# B&R Automation Studio project NAEUL004C00R13L518F00 (part 36)

#### Act_InputConfig.st
```iecst
ACTION Act_InputConfig:

	pa_tyMpProdRcp ACCESS p_ProdRcpCurrList; // Accessing the Current Product Recipe List

	tylocalMpProdRcp.In.udiRstErr := g_tyRstErrOut.udiRstErr;
	tylocalMpProdRcp.In.sPVName	  := g_tyNtParamCurr.sMpProdRcpPVNm;
	tylocalMpProdRcp.In.sFileName := g_tyNtParamCurr.sMpProdRcpFileNm;
	tylocalMpProdRcp.In.sProgNm   := g_tyNtParamCurr.sProdRcpProgNm;

	IF g_tyStartUp.bRun THEN
		tylocalMpProdRcp.In.eAct := g_tyStartUp.eMpProdRcpAct;
	ELSE
		tylocalMpProdRcp.In.eAct := g_tyUIOut.eMnlAct.eMpProdRcpAct;
	END_IF

END_ACTION
```

#### Act_Main.st
```iecst
ACTION Act_Main:

	//Set p_eAct
	IF tylocalMpProdRcp.Out.eStatus = Idle THEN
		tylocalMpProdRcp.Out.eStat	:= tylocalMpProdRcp.In.eAct;
	END_IF

	//Main
	CASE tylocalMpProdRcp.Out.eStat OF

		MpProdRcpActIdle:
			IF tylocalMpProdRcp.Out.eStatus <> Idle THEN	//Reset Data
				//Private
				fbDirCreate1(bEn := FALSE);
				fbDirCreate2(bEn := FALSE);
				fbMpRecipeRegPar(Enable := FALSE);
				fbMpRecipeXml(Enable := FALSE);
				usiStep			:= 0;

				sStatTxt	:= a_sStatText[tylocalMpProdRcp.Out.eStat];

			END_IF

			tylocalMpProdRcp.Out.eStatus	:= Idle;

		MpProdRcpActCreateDir:
			IF tylocalMpProdRcp.Out.eStatus = Idle OR tylocalMpProdRcp.Out.eStatus = Busy THEN

				tylocalMpProdRcp.Out.eStatus	:= Busy;

				sStatTxt	:= a_sStatText[tylocalMpProdRcp.Out.eStat];

				CASE usiStep OF
					0:
						fbDirCreate1(bEn := TRUE);
						IF fbDirCreate1.udiStatus = 0 THEN
							usiStep	:= 1;
						ELSIF fbDirCreate1.udiStatus < 65534 THEN
							tylocalMpProdRcp.Out.eStatus		:= Error;

							IF fbDirCreate1.udiStatus = 1908 THEN
								udiStatus	:= 10000;	//Create User Directory Error
							ELSE
								udiStatus	:= fbDirCreate1.udiStatus;
							END_IF
						END_IF

					1:
						fbDirCreate2(bEn := TRUE);
						IF fbDirCreate2.udiStatus = 0 THEN
							tylocalMpProdRcp.Out.eStatus	:= Done;
						ELSIF fbDirCreate2.udiStatus < 65534 THEN
							tylocalMpProdRcp.Out.eStatus		:= Error;

							IF fbDirCreate2.udiStatus = 1908 THEN
								udiStatus	:= 10001;	//Create Product Recipe Directory Error
							ELSE
								udiStatus	:= fbDirCreate2.udiStatus;
							END_IF
						END_IF

				END_CASE

			END_IF

		MpProdRcpActLoad:
			IF tylocalMpProdRcp.Out.eStatus = Idle OR tylocalMpProdRcp.Out.eStatus = Busy THEN

				tylocalMpProdRcp.Out.eStatus	:= Busy;

				sStatTxt	:= a_sStatText[tylocalMpProdRcp.Out.eStat];

				CASE usiStep OF
					0:
						fbMpRecipeRegPar(Enable := TRUE);

						IF (fbMpRecipeRegPar.Active = TRUE) AND (fbMpRecipeRegPar.StatusID = 0) THEN
							usiStep	:= 1;
						ELSIF fbMpRecipeRegPar.StatusID <> 0 THEN
							tylocalMpProdRcp.Out.eStatus		:= Error;
							udiStatus	:= 10002;	//MpRecipeRegPar Error While Loading
						END_IF

					1:
						fbMpRecipeXml.Load	:= TRUE;
						fbMpRecipeXml.Save	:= FALSE;
						fbMpRecipeXml(Enable := TRUE);

						IF (fbMpRecipeXml.Active = TRUE) AND (fbMpRecipeXml.CommandDone = TRUE) AND (fbMpRecipeXml.StatusID = 0) THEN
							tylocalMpProdRcp.Out.eStatus	:= Done;
							pa_tyMpProdRcp	:= a_tyMpProdRcp1;
						ELSIF fbMpRecipeXml.StatusID <> 0 THEN
							tylocalMpProdRcp.Out.eStatus		:= Error;
							udiStatus	:= 10003;	//MpRecipeXml Error While Loading
						END_IF

				END_CASE

			END_IF

		MpProdRcpActSave:
			IF tylocalMpProdRcp.Out.eStatus = Idle OR tylocalMpProdRcp.Out.eStatus = Busy THEN

				tylocalMpProdRcp.Out.eStatus	:= Busy;

				sStatTxt	:= a_sStatText[tylocalMpProdRcp.Out.eStat];

				CASE usiStep OF
					0:
						a_tyMpProdRcp1	:= pa_tyMpProdRcp;
						fbMpRecipeRegPar(Enable := TRUE);

						IF (fbMpRecipeRegPar.Active = TRUE) AND (fbMpRecipeRegPar.StatusID = 0) THEN
							usiStep	:= 1;
						ELSIF fbMpRecipeRegPar.StatusID <> 0 THEN
							tylocalMpProdRcp.Out.eStatus		:= Error;
							udiStatus	:= 10004;	//MpRecipeRegPar Error While Saving
						END_IF

					1:
						fbMpRecipeXml.Load	:= FALSE;
						fbMpRecipeXml.Save	:= TRUE;
						fbMpRecipeXml(Enable := TRUE);

						IF (fbMpRecipeXml.Active = TRUE) AND (fbMpRecipeXml.CommandDone = TRUE) AND (fbMpRecipeXml.StatusID = 0) THEN
							tylocalMpProdRcp.Out.eStatus	:= Done;
						ELSIF fbMpRecipeXml.StatusID <> 0 THEN
							tylocalMpProdRcp.Out.eStatus		:= Error;
							udiStatus	:= 10005;	//MpRecipeXml Error While Saving
						END_IF

				END_CASE

			END_IF

	END_CASE

END_ACTION
```

#### Act_OutputConfig.st
```iecst
ACTION Act_OutputConfig:

	g_tyMpProdRcp	:= tylocalMpProdRcp.Out;

END_ACTION
```

#### Cyclic.st
```iecst
PROGRAM _CYCLIC

	IF bInitialDone = FALSE THEN
		IF g_tyStartUp.bNtSettingsLoadDone = TRUE THEN
			bInitialDone	:= TRUE;
			Act_Initial;
		END_IF

	ELSE

		Act_InputConfig;
		Act_Main;
		Act_OutputConfig;
		Act_Alarm;

	END_IF

END_PROGRAM
```

### Package Logical/MagRcp - pending

### MagRcp.typ - Change By Project
```iecst
(*2020-07-24*)
(**)
(*Action*)

TYPE
	eMagRcpAction :
		(
		MagRcpActIdle,
		MagRcpActCreateDir,
		MagRcpActAddEdit,
		MagRcpActDel,
		MagRcpActGetInfo,
		MagRcpActGetList,
		MagRcpActFilter,
		MagRcpActReadCurrRcp,
		MagRcpActLoadRcp,
		MagRcpActWriteCurrRcpParam,
		MagRcpActSaveList,
		MagRcpActSort
		);
END_TYPE

(**)
(*Data*)

TYPE
	tyMagRcpParam : 	STRUCT
		sRcpNm : STRING[30];
		diTtlSlt : DINT;
		diSltToSltInUM : DINT;
		diMag1Slt1PosInUM : DINT;
		diMag2Slt1PosInUM : DINT;
		diMag3Slt1PosInUM : DINT;
		diMag1TravPosInUM : DINT;
		diMag2TravPosInUM : DINT;
		diMag3TravPosInUM : DINT;
		usiMagModel : USINT;
		sDisplayInfo : STRING[30];
		diMagMaxBrdWidth : DINT;
		dtLastModified : DATE_AND_TIME;
		bSafetyBarDisabled : BOOL;
		bMagHeightChkEn : BOOL;
	END_STRUCT;
END_TYPE
```

### MagRcp.var - Change By Project
```iecst
(*2020-07-24*)
(**)
(*Constant*)
VAR CONSTANT
	c_udiMagRcpMax : UDINT := 10;
END_VAR
(**)
(*Action & State & Status*)
VAR
	p_MagRcpStat : UDINT;
	p_MagRcpStatus : UDINT;
	p_MagRcpStatTxt : UDINT;
END_VAR
(**)
(*Alarm*)
VAR
	p_MagRcpAlmData : UDINT;
END_VAR
(**)
(*Output*)
VAR
	p_MagRcpNmExist : UDINT;
	p_MagRcpNmNotExist : UDINT;
	p_MagRcpNmEmpty : UDINT;
	p_MagRcpListFull : UDINT;
	p_MagRcpCurrList : UDINT;
	p_MagRcpFilterList : UDINT;
	p_MagRcpSortedList : UDINT;
	p_MagRcpInfoOut : UDINT;
	p_MagRcpFileNotFound : UDINT;
	p_MagRcpCurrRcp : UDINT;
	p_MagRcpCurrRcpNm : UDINT;
	p_MagRcpCurrRcpTtlSlt : UDINT;
	p_MagRcpCurrRcpSltToSlt : UDINT;
	p_MagRcpCurrRcpMag1Slt1Pos : UDINT;
	p_MagRcpCurrRcpMag2Slt1Pos : UDINT;
	p_MagRcpCurrRcpMag3Slt1Pos : UDINT;
	p_MagRcpCurrRcpMag1TravPos : UDINT;
	p_MagRcpCurrRcpMag2TravPos : UDINT;
	p_MagRcpCurrRcpMag3TravPos : UDINT;
	p_MagRcpCurrRcpDisplayInfo : UDINT;
	p_MagRcpCurrRcpMagMaxBrdWidth : UDINT;
	p_MagRcpCurrRcpLastModified : UDINT;
	p_MagRcpCurrRcpMagModel : UDINT;
	p_MagRcpCurrRcpSBarDisabled : UDINT;
	p_MagRcpCurrRcpMagHeightChkEn : UDINT;
END_VAR
(**)
```

### Program Logical/MagRcp/MagRcp (IEC) - 1.00.0 - NtRecipe v5.00.0 , NtFileIO v5.00.0

#### InputRef.var
```iecst
(*2019-05-07*)
(**)
(*General*)
VAR
	p_eAct : REFERENCE TO eMagRcpAction;
	p_udiMax : REFERENCE TO UDINT;
	p_udiRstErr : REFERENCE TO UDINT;
	p_bPrep : REFERENCE TO BOOL;
	p_bDis : REFERENCE TO BOOL;
END_VAR
(**)
(*Configuration*)
VAR
	p_dtCurrDT : REFERENCE TO DATE_AND_TIME;
	p_sSearch : REFERENCE TO STRING[30];
	p_tyInfoIn : REFERENCE TO tyMagRcpParam;
	p_tyCurrRcpWr : REFERENCE TO tyMagRcpParam;
	p_sListFileName : REFERENCE TO STRING[80];
	p_sSingleFileName : REFERENCE TO STRING[80];
	p_sProgNm : REFERENCE TO STRING[15];
	p_bNtSettingsLoadDone : REFERENCE TO BOOL;
	p_eLinkLCSMngRcpMagRcpAct : REFERENCE TO eMagRcpAction;
	p_bLinkNtParamLCSManageRcpPrep : REFERENCE TO BOOL;
	p_bLinkMcParamLCSManageRcpEn : REFERENCE TO BOOL;
	p_eLinkUIMagRcpAct : REFERENCE TO eMagRcpAction;
END_VAR
```

#### InputRef_Link.var
```iecst
(*2019-03-25*)
(**)
VAR
	rSltToSlt : REAL;
	sSltToSlt : STRING[30];
	sTtlSlt : STRING[30];
	p_bLinkStartupRun : REFERENCE TO BOOL;
END_VAR
```

#### Local.var
```iecst
(*2019-05-09*)
(**)
(*Local Action, State & Status*)
VAR
	eAct : eMagRcpAction := MagRcpActIdle;
	eStat : eMagRcpAction := MagRcpActIdle;
	eStatus : eFBStatus := Idle;
	udiStatus : UDINT := 0;
	sStatTxt : STRING[200] := '';
	a_sStatText : ARRAY[0..50] OF STRING[200] := ['Idling','Creating Directory','Adding and Editing Files','Deleting Files','Get Info','Get List','Filtering Files','Reading Current Recipe','Loading Current Recipe','Writing Current Recipe Parameter','Saving List',40('')];
END_VAR
(**)
(*Local Alarm*)
VAR
	tyAlmData : tyAlmDat;
	a_tyAlmText : ARRAY[10000..10099] OF tyAlmTxt := [(sAlmText:='Create User Directory Error',sRcyText:='Unable To Create User Directory. Please Contact Nutek For A Possible Solution'),(sAlmText:='Create Magazine Recipe Directory Error',sRcyText:='Unable To Create Magazine Recipe Directory. Please Contact Nutek For A Possible Solution'),(sAlmText:='File Open Error While Adding & Editing',sRcyText:='An Error Was Encountered While Trying To Open File. Please Contact Nutek For A Possible Solution.'),(sAlmText:='File Create Error While Adding & Editing',sRcyText:='An Error Was Encountered While Trying To Create File. Please Contact Nutek For A Possible Solution.'),(sAlmText:='File Write Error While Adding & Editing',sRcyText:='An Error Was Encountered While Trying To Write File. Please Contact Nutek For A Possible Solution.'),(sAlmText:='File Close Error While Adding & Editing',sRcyText:='An Error Was Encountered While Trying To Close File. Please Contact Nutek For A Possible Solution.'),(sAlmText:='File Open Error While Deleting',sRcyText:='An Error Was Encountered While Trying To Open File. Please Contact Nutek For A Possible Solution.'),(sAlmText:='File Create Error While Deleting',sRcyText:='An Error Was Encountered While Trying To Create File. Please Contact Nutek For A Possible Solution.'),(sAlmText:='File Write Error While Deleting',sRcyText:='An Error Was Encountered While Trying To Write File. Please Contact Nutek For A Possible Solution.'),(sAlmText:='File Close Error While Deleting',sRcyText:='An Error Was Encountered While Trying To Close File. Please Contact Nutek For A Possible Solution.'),(sAlmText:='File Open Error While Getting List',sRcyText:='An Error Was Encountered While Trying To Open File. Please Contact Nutek For A Possible Solution.'),(sAlmText:='File Read Error While Getting List',sRcyText:='An Error Was Encountered While Trying To Read File. Please Contact Nutek For A Possible Solution.'),(sAlmText:='File Close Error While Getting List',sRcyText:='An Error Was Encountered While Trying To Close File. Please Contact Nutek For A Possible Solution.'),(sAlmText:='Directory Does Not Exist While Adding & Editing',sRcyText:='The Directory Does Not Exist.Please Contact Nutek For A Possible Solution.'),(sAlmText:='Directory Does Not Exist While Deleting',sRcyText:='The Directory Does Not Exist.Please Contact Nutek For A Possible Solution.'),(sAlmText:='File Open Error While Loading Current Recipe',sRcyText:='An Error Was Encountered While Trying To Open File. Please Contact Nutek For A Possible Solution.'),(sAlmText:='File Create Error While Loading Current Recipe',sRcyText:='An Error Was Encountered While Trying To Create File. Please Contact Nutek For A Possible Solution.'),(sAlmText:='File Write Error While Loading Current Recipe',sRcyText:='An Error Was Encountered While Trying To Write File. Please Contact Nutek For A Possible Solution.'),(sAlmText:='File Close Error While Loading Current Recipe',sRcyText:='An Error Was Encountered While Trying To Close File. Please Contact Nutek For A Possible Solution.'),(sAlmText:='Directory Does Not Exist While Loading Current Recipe',sRcyText:='The Directory Does Not Exist.Please Contact Nutek For A Possible Solution.'),(sAlmText:='File Open Error While Reading Current Recipe',sRcyText:='An Error Was Encountered While Trying To Open File. Please Contact Nutek For A Possible Solution.'),(sAlmText:='File Read Error While Reading Current Recipe',sRcyText:='An Error Was Encountered While Trying To Read File. Please Contact Nutek For A Possible Solution.'),(sAlmText:='File Close Error While Reading Current Recipe',sRcyText:='An Error Was Encountered While Trying To Close File. Please Contact Nutek For A Possible Solution.'),(sAlmText:='File Open Error While Writing Current Recipe Parameter',sRcyText:='An Error Was Encountered While Trying To Open File. Please Contact Nutek For A Possible Solution.'),(sAlmText:='File Create Error While Writing Current Recipe Parameter',sRcyText:='An Error Was Encountered While Trying To Create File. Please Contact Nutek For A Possible Solution.'),(sAlmText:='File Write Error While Writing Current Recipe Parameter',sRcyText:='An Error Was Encountered While Trying To Write File. Please Contact Nutek For A Possible Solution.'),(sAlmText:='File Close Error While Writing Current Recipe Parameter',sRcyText:='An Error Was Encountered While Trying To Close File. Please Contact Nutek For A Possible Solution.'),(sAlmText:='Directory Does Not Exist While Writing Current Recipe Parameter',sRcyText:='The Directory Does Not Exist.Please Contact Nutek For A Possible Solution.'),(sAlmText:='File Open Error While Saving List',sRcyText:='An Error Was Encountered While Trying To Open File. Please Contact Nutek For A Possible Solution.'),(sAlmText:='File Create Error While Saving List',sRcyText:='An Error Was Encountered While Trying To Create File. Please Contact Nutek For A Possible Solution.'),(sAlmText:='File Write Error While Saving List',sRcyText:='An Error Was Encountered While Trying To Write File. Please Contact Nutek For A Possible Solution.'),(sAlmText:='File Close Error While Saving List',sRcyText:='An Error Was Encountered While Trying To Close File. Please Contact Nutek For A Possible Solution.'),(sAlmText:='Directory Does Not Exist While Saving List',sRcyText:='The Directory Does Not Exist.Please Contact Nutek For A Possible Solution.'),67(0)];
END_VAR
(**)
(*Local Output*)
VAR
	bNmExist : BOOL;
	bNmNotExist : BOOL;
	bNmEmpty : BOOL;
	bListFull : BOOL;
	a_tyCurrList : ARRAY[1..c_udiMagRcpMax] OF tyMagRcpParam;
	a_tyFilterList : ARRAY[1..c_udiMagRcpMax] OF tyMagRcpParam;
	a_tySortList : ARRAY[1..c_udiMagRcpMax] OF tyMagRcpParam;
	tyTempList : tyMagRcpParam;
	tyInfoOut : tyMagRcpParam;
	bFileNotFound : BOOL;
	tyCurrRcp : tyMagRcpParam;
END_VAR
(**)
(*Local Input*)
VAR
	udiRstErr : UDINT := 0;
	bPrep : BOOL := TRUE;
	bDis : BOOL := FALSE;
	dtCurrDT : DATE_AND_TIME;
	sSearch : STRING[30] := '';
	tyInfoIn : tyMagRcpParam;
	tyCurrRcpWr : tyMagRcpParam;
	sListFileName : STRING[80] := 'MagazineRecipeList.dat';
	sSingleFileName : STRING[80] := 'MagazineRecipe.dat';
	sProgNm : STRING[15] := 'MagRcp';
	bNtSettingsLoadDone : BOOL := TRUE;
	udiSortCurrenTotalCntr : UDINT;
	iSortCurrentInnerCntr : INT;
	iSortCurrentOuterCntr : INT;
	iTotalRcp : INT;
	i : {REDUND_UNREPLICABLE} INT;
	udi : UDINT;
	sDebug : STRING[300];
	tyTempRecipe : tyMagRcpParam;
END_VAR
(**)
(*Local*)
VAR
	bRstErr : BOOL;
	udiRstErrOld : UDINT;
	bInitDone : BOOL;
	bInitialDone : BOOL;
	usiStep : USINT;
	udiAddStatus : UDINT;
	a_tyListTemp : ARRAY[1..c_udiMagRcpMax] OF tyMagRcpParam;
	fbDirCreate1 : fbDirCreate;
	fbDirCreate2 : fbDirCreate;
	fbFileReadList : fbFileFullRead;
	fbFileWriteList : fbFileFullWrite;
	fbFileReadSingle : fbFileFullRead;
	fbFileWriteSingle : fbFileFullWrite;
	fbFileLoadSingle : fbFileFullWrite;
	iFilterCtr : INT;
	udiModuleNum : UDINT := 4901;
END_VAR
```

#### Act_Action.st
```iecst
(** 2019-03-25 **)
ACTION Act_Action:

	//Reset Error
	IF (eStatus = Error) AND bRstErr THEN
		p_eAct	:= MagRcpActIdle;
		eStat	:= MagRcpActIdle;
	END_IF

	//Reset Done
	IF eStatus = Done AND p_eAct = MagRcpActIdle THEN
		eStat	:= MagRcpActIdle;
	END_IF

	//Set p_eAct
	IF eStatus = Idle THEN
		eStat	:= p_eAct;
	END_IF

END_ACTION
```

#### Act_Alarm.st
```iecst
(** 2019-03-25 **)
ACTION Act_Alarm:

	//Error
	IF EDGEPOS(eStatus = Error) THEN

		tyAlmData.sProgNm		:= p_sProgNm;
		tyAlmData.udiCode		:= udiStatus;
		tyAlmData.eSeverity		:= AlmSeverityError;
		tyAlmData.udiRunTime	:= tyAlmData.udiRunTime + 1;
		tyAlmData.bAlm			:= TRUE;
		tyAlmData.udiModuleNum  := udiModuleNum;
		g_sMagRcpProgNm			:= p_sProgNm;

		//Get Error Message
		IF tyAlmData.udiCode < 10000 OR tyAlmData.udiCode > 10099 THEN
			tyAlmData.sAlmMsg	:= 'Unknown';
			tyAlmData.sRcyMsg	:= 'Unknown';
		ELSE
			tyAlmData.sAlmMsg	:= a_tyAlmText[tyAlmData.udiCode].sAlmText;
			tyAlmData.sRcyMsg	:= a_tyAlmText[tyAlmData.udiCode].sRcyText;
		END_IF

		sStatTxt	:= tyAlmData.sAlmMsg;

	ELSIF bRstErr AND (tyAlmData.udiCode <> 0) THEN

		tyAlmData.udiCode	:= 0;
		tyAlmData.eSeverity	:= AlmSeverityNA;
		tyAlmData.sAlmMsg	:= '';
		tyAlmData.sRcyMsg	:= '';
		tyAlmData.bAlm			:= FALSE;
		sStatTxt	:= a_sStatText[eStat];

	END_IF

END_ACTION
```

#### Act_InitGlobal.st
```iecst
(** 2019-03-25 **)
ACTION Act_InitGlobal:

	(* Always Change If Project Change *)

	//Pass Data To Link
	p_bLinkStartupRun ACCESS p_StartupRun;

	//Pass Data To Internal Use
	p_udiRstErr ACCESS p_RstErrReset;
	p_dtCurrDT ACCESS p_TimeCurrDT;
	p_sSearch ACCESS p_UIMagRcpSearch;
	//p_tyInfoIn ACCESS p_UIMagRcpInfoIn;
	p_sListFileName ACCESS p_NtParamMagRcpListFileNm;
	p_sSingleFileName ACCESS p_NtParamMagRcpSingleFileNm;
	p_sProgNm ACCESS p_NtParamMagRcpProgNm;
	p_bNtSettingsLoadDone ACCESS p_StartupNtSettingsLoadDone;
	p_eLinkLCSMngRcpMagRcpAct ACCESS p_LCSMngRcpMagRcpAct;
	p_bLinkNtParamLCSManageRcpPrep ACCESS p_NtParamLCSManageRcpPrep;
	p_bLinkMcParamLCSManageRcpEn ACCESS p_McParamLCSManageRcpEn;
	p_eLinkUIMagRcpAct ACCESS p_UIMagRcpAct;
	(* Always Change If Project Change *)

END_ACTION
```

#### Act_Initial.st
```iecst
(** 2019-05-07 **)
ACTION Act_Initial:

	//Initial
	sStatTxt	:= a_sStatText[eStat];

	fbDirCreate1.sDevice	:= 'F';
	fbDirCreate1.sDirName	:= 'User';
	fbDirCreate1(bEn := FALSE);

	fbDirCreate2.sDevice	:= 'User';
	fbDirCreate2.sDirName	:= 'MagazineRecipe';
	fbDirCreate2(bEn := FALSE);

	fbFileReadList.sDevice			:= 'MagRcp';
	fbFileReadList.sFile			:= p_sListFileName;
	fbFileReadList.udiOffset		:= 0;
	fbFileReadList.p_Dest			:= ADR(a_tyCurrList);
	fbFileReadList.udiLen			:= SIZEOF(a_tyCurrList);
	fbFileReadList(bEn := FALSE);

	fbFileWriteList.sDevice			:= 'MagRcp';
	fbFileWriteList.sFile			:= p_sListFileName;
	fbFileWriteList.udiOffset		:= 0;
	fbFileWriteList.p_Src			:= ADR(a_tyListTemp);
	fbFileWriteList.udiLen			:= SIZEOF(a_tyListTemp);
	fbFileWriteList.udiOption		:= 0;
	fbFileWriteList(bEn := FALSE);

	fbFileReadSingle.sDevice		:= 'MagRcp';
	fbFileReadSingle.sFile			:= p_sSingleFileName;
	fbFileReadSingle.udiOffset		:= 0;
	fbFileReadSingle.p_Dest			:= ADR(tyCurrRcp);
	fbFileReadSingle.udiLen			:= SIZEOF(tyCurrRcp);
	fbFileReadSingle(bEn := FALSE);

	fbFileLoadSingle.sDevice		:= 'MagRcp';
	fbFileLoadSingle.sFile			:= p_sSingleFileName;
	fbFileLoadSingle.udiOffset		:= 0;
	fbFileLoadSingle.p_Src			:= ADR(tyCurrRcp);
	fbFileLoadSingle.udiLen			:= SIZEOF(tyCurrRcp);
	fbFileLoadSingle.udiOption		:= 0;
	fbFileLoadSingle(bEn := FALSE);

	fbFileWriteSingle.sDevice		:= 'MagRcp';
	fbFileWriteSingle.sFile			:= p_sSingleFileName;
	fbFileWriteSingle.udiOffset		:= 0;
	fbFileWriteSingle.p_Src			:= ADR(p_tyCurrRcpWr);
	fbFileWriteSingle.udiLen		:= SIZEOF(p_tyCurrRcpWr);
	fbFileWriteSingle.udiOption		:= 0;
	fbFileWriteSingle(bEn := FALSE);

END_ACTION
```

#### Act_InitLocal.st
```iecst
(** 2019-05-07 **)
ACTION Act_InitLocal:

	//Input Reference Link To Local Variable
	p_eAct ACCESS ADR(eAct);
	p_udiMax ACCESS ADR(c_udiMagRcpMax);
	p_udiRstErr ACCESS ADR(udiRstErr);
	p_bPrep ACCESS ADR(bPrep);
	p_bDis ACCESS ADR(bDis);
	p_dtCurrDT ACCESS ADR(dtCurrDT);
	p_sSearch ACCESS ADR(sSearch);
	p_tyInfoIn ACCESS ADR(tyInfoIn);
	p_tyCurrRcpWr ACCESS ADR(tyCurrRcpWr);
	p_sListFileName ACCESS ADR(sListFileName);
	p_sSingleFileName ACCESS ADR(sSingleFileName);
	p_sProgNm ACCESS ADR(sProgNm);
	p_bNtSettingsLoadDone ACCESS ADR(bNtSettingsLoadDone);

END_ACTION
```

#### Act_Link.st
```iecst
(** 2019-03-29 **)
ACTION Act_Link:

	IF p_eAct = MagRcpActAddEdit THEN

		rSltToSlt	:= DINT_TO_REAL(p_tyInfoIn.diSltToSltInUM);
		rSltToSlt	:= rSltToSlt / 1000;
		sSltToSlt	:= REAL_TO_STRING(rSltToSlt);
		sTtlSlt		:= DINT_TO_STRING(p_tyInfoIn.diTtlSlt);

		p_tyInfoIn.sDisplayInfo	:= sSltToSlt;
		p_tyInfoIn.sDisplayInfo	:= CONCAT(p_tyInfoIn.sDisplayInfo , ' | ');
		p_tyInfoIn.sDisplayInfo	:= CONCAT(p_tyInfoIn.sDisplayInfo , sTtlSlt);

	END_IF

END_ACTION
```

#### Act_LinkAction.st
```iecst
(** 2019-03-29 **)
ACTION Act_LinkAction:

	IF p_bLinkStartupRun = TRUE THEN
		p_eAct ACCESS p_StartupMagRcpAct;
	ELSE

		IF p_bLinkNtParamLCSManageRcpPrep AND p_bLinkMcParamLCSManageRcpEn THEN
			IF p_eLinkLCSMngRcpMagRcpAct <> MagRcpActIdle THEN
				p_eAct ACCESS p_LCSMngRcpMagRcpAct;
				p_tyInfoIn ACCESS p_LCSMngRcpMagRcpInfoIn;
			ELSIF p_eLinkUIMagRcpAct <> MagRcpActIdle THEN
				p_eAct ACCESS p_UIMagRcpAct;
				p_tyInfoIn ACCESS p_UIMagRcpInfoIn;

				p_tyInfoIn.dtLastModified	:= p_dtCurrDT;
			END_IF
		ELSE
			p_eAct ACCESS p_UIMagRcpAct;
			p_tyInfoIn ACCESS p_UIMagRcpInfoIn;

			p_tyInfoIn.dtLastModified	:= p_dtCurrDT;
		END_IF
	END_IF

END_ACTION
```

#### Act_Main.st
```iecst
(** 2019-05-09 **)
ACTION Act_Main:

	//Main
	CASE eStat OF

		MagRcpActIdle:
			IF eStatus <> Idle THEN	//Reset Data
				//Private
				fbDirCreate1(bEn := FALSE);
				fbDirCreate2(bEn := FALSE);
				fbFileReadList(bEn := FALSE);
				fbFileWriteList(bEn := FALSE);
				fbFileReadSingle(bEn := FALSE);
				fbFileWriteSingle(bEn := FALSE);
				fbFileLoadSingle(bEn := FALSE);
				usiStep			:= 0;
				udiAddStatus	:= 0;

				bNmExist		:= FALSE;
				bNmNotExist		:= FALSE;
				bNmEmpty		:= FALSE;
				bListFull		:= FALSE;
				bFileNotFound	:= FALSE;
				iTotalRcp		:= 0;

				memset(ADR(tyTempRecipe), 0 , SIZEOF(tyTempRecipe));

				sStatTxt	:= a_sStatText[eStat];

			END_IF

			eStatus	:= Idle;

		MagRcpActCreateDir:
			IF eStatus = Idle OR eStatus = Busy THEN

				eStatus	:= Busy;

				sStatTxt	:= a_sStatText[eStat];

				CASE usiStep OF
					0:
						fbDirCreate1(bEn := TRUE);
						IF fbDirCreate1.udiStatus = 0 THEN
							usiStep	:= 1;
						ELSIF fbDirCreate1.udiStatus < 65534 THEN
							eStatus		:= Error;

							IF fbDirCreate1.udiStatus = 1908 THEN
								udiStatus	:= 10000;	//Create User Directory Error
							ELSE
								udiStatus	:= fbDirCreate1.udiStatus;
							END_IF
						END_IF

					1:
						fbDirCreate2(bEn := TRUE);
						IF fbDirCreate2.udiStatus = 0 THEN
							eStatus	:= Done;
						ELSIF fbDirCreate2.udiStatus < 65534 THEN
							eStatus		:= Error;

							IF fbDirCreate2.udiStatus = 1908 THEN
								udiStatus	:= 10001;	//Create Magazine Recipe Directory Error
							ELSE
								udiStatus	:= fbDirCreate2.udiStatus;
							END_IF
						END_IF

				END_CASE

			END_IF

		MagRcpActAddEdit:
			IF eStatus = Idle OR eStatus = Busy THEN

				eStatus	:= Busy;

				sStatTxt	:= a_sStatText[eStat];

				CASE usiStep OF
					0:	//Edit Recipe
						udiAddStatus	:= fRecipeAddEdit(ADR(p_tyInfoIn) , ADR(a_tyListTemp) , SIZEOF(a_tyListTemp[1]) , ADR(a_tyListTemp[1].sRcpNm) , SIZEOF(a_tyListTemp[1].sRcpNm) , p_udiMax);

						IF udiAddStatus = 1600 THEN	//Recipe Name Empty
							bNmEmpty	:= TRUE;
							eStatus		:= Done;

						ELSIF udiAddStatus = 1601 THEN	//Recipe Full
							bListFull	:= TRUE;
							eStatus		:= Done;

						ELSIF udiAddStatus = 0 THEN	//OK
							usiStep	:= 1;

						END_IF

					1:	//Write Into File
						fbFileWriteList(bEn := TRUE);

						IF fbFileWriteList.udiStatus = 0 THEN
							a_tyCurrList	:= a_tyListTemp;
							eStatus			:= Done;

						ELSIF fbFileWriteList.udiStatus < 65534 THEN
							a_tyListTemp	:= a_tyCurrList;
							eStatus			:= Error;

							IF fbFileWriteList.udiStatus = 1900 THEN
								udiStatus	:= 10002;	//File Open Error While Adding & Editing
							ELSIF fbFileWriteList.udiStatus = 1901 THEN
								udiStatus	:= 10003;	//File Create Error While Adding & Editing
							ELSIF fbFileWriteList.udiStatus = 1903 THEN
								udiStatus	:= 10004;	//File Write Error While Adding & Editing
							ELSIF fbFileWriteList.udiStatus = 1904 THEN
								udiStatus	:= 10005;	//File Close Error While Adding & Editing
							ELSIF fbFileWriteList.udiStatus = 1914 THEN
								udiStatus	:= 10013;	//Directory Does Not Exist While Adding & Editing
							ELSE
								udiStatus	:= fbFileWriteList.udiStatus;
							END_IF
						END_IF

				END_CASE

			END_IF

		MagRcpActDel:
			IF eStatus = Idle OR eStatus = Busy THEN

				eStatus	:= Busy;

				sStatTxt	:= a_sStatText[eStat];

				CASE usiStep OF
					0:	//Delete Recipe
						udiAddStatus	:= fRecipeDelete(ADR(p_tyInfoIn) , ADR(a_tyListTemp) , SIZEOF(a_tyListTemp[1]) , ADR(a_tyListTemp[1].sRcpNm) , SIZEOF(a_tyListTemp[1].sRcpNm) , p_udiMax);

						IF udiAddStatus = 1600 THEN	//Recipe Name Empty
							bNmEmpty	:= TRUE;
							eStatus		:= Done;

						ELSIF udiAddStatus = 1603 THEN	//Recipe Not Exist
							bNmNotExist	:= TRUE;
							eStatus		:= Done;

						ELSIF udiAddStatus = 0 THEN	//OK
							usiStep	:= 1;

						END_IF

					1:	//Write Into File
						fbFileWriteList(bEn := TRUE);

						IF fbFileWriteList.udiStatus = 0 THEN
							a_tyCurrList	:= a_tyListTemp;
							eStatus			:= Done;

						ELSIF fbFileWriteList.udiStatus < 65534 THEN
							a_tyListTemp	:= a_tyCurrList;
							eStatus			:= Error;

							IF fbFileWriteList.udiStatus = 1900 THEN
								udiStatus	:= 10006;	//File Open Error While Deleting
							ELSIF fbFileWriteList.udiStatus = 1901 THEN
								udiStatus	:= 10007;	//File Create Error While Deleting
							ELSIF fbFileWriteList.udiStatus = 1903 THEN
								udiStatus	:= 10008;	//File Write Error While Deleting
							ELSIF fbFileWriteList.udiStatus = 1904 THEN
								udiStatus	:= 10009;	//File Close Error While Deleting
							ELSIF fbFileWriteList.udiStatus = 1914 THEN
								udiStatus	:= 10014;	//Directory Does Not Exist While Deleting
							ELSE
								udiStatus	:= fbFileWriteList.udiStatus;
							END_IF
						END_IF

				END_CASE

			END_IF

		MagRcpActGetInfo:
			IF eStatus = Idle OR eStatus = Busy THEN

				sStatTxt	:= a_sStatText[eStat];

				IF p_tyInfoIn.sRcpNm = '' THEN
					bNmEmpty	:= TRUE;
					bNmNotExist	:= TRUE;
				ELSE
					bNmNotExist	:= (fRecipeGetInfo(p_tyInfoIn.sRcpNm , ADR(tyInfoOut) , ADR(a_tyCurrList) , SIZEOF(a_tyCurrList[1]) , ADR(a_tyCurrList[1].sRcpNm) , SIZEOF(a_tyCurrList[1].sRcpNm) , p_udiMax)) = 0;
				END_IF

				eStatus	:= Done;

			END_IF

		MagRcpActGetList:
			IF eStatus = Idle OR eStatus = Busy THEN

				eStatus	:= Busy;

				sStatTxt	:= a_sStatText[eStat];

				fbFileReadList(bEn := TRUE);
				IF fbFileReadList.udiStatus = 0 THEN
					a_tyListTemp	:= a_tyCurrList;
					eStatus			:= Done;

				ELSIF fbFileReadList.udiStatus < 65534 THEN
					eStatus		:= Error;

					IF fbFileReadList.udiStatus = 1900 THEN
						udiStatus	:= 10010;	//File Open Error While Getting List
					ELSIF fbFileReadList.udiStatus = 1902 THEN
						udiStatus	:= 10011;	//File Read Error While Getting List
					ELSIF fbFileReadList.udiStatus = 1904 THEN
						udiStatus	:= 10012;	//File Close Error While Getting List
					ELSIF fbFileReadList.udiStatus = 1915 THEN
						bFileNotFound	:= TRUE;
						eStatus			:= Done;
					ELSE
						udiStatus	:= fbFileReadList.udiStatus;
					END_IF
				END_IF

			END_IF

		MagRcpActFilter:
			IF eStatus = Idle OR eStatus = Busy THEN

				sStatTxt	:= a_sStatText[eStat];

				CASE usiStep OF
					0:
						fRecipeFilter(p_sSearch , ADR(a_tyFilterList) , ADR(a_tyCurrList) , SIZEOF(a_tyCurrList[1]) , ADR(a_tyCurrList[1].sRcpNm) ,
						SIZEOF(a_tyCurrList[1].sRcpNm) , p_udiMax, 0, 499, iFilterCtr);
						usiStep := 1;
					1:
						fRecipeFilter(p_sSearch , ADR(a_tyFilterList) , ADR(a_tyCurrList) , SIZEOF(a_tyCurrList[1]) , ADR(a_tyCurrList[1].sRcpNm) ,
						SIZEOF(a_tyCurrList[1].sRcpNm) , p_udiMax, 500, 999, iFilterCtr);
						usiStep := 2;
					2:
						fRecipeFilter(p_sSearch , ADR(a_tyFilterList) , ADR(a_tyCurrList) , SIZEOF(a_tyCurrList[1]) , ADR(a_tyCurrList[1].sRcpNm) ,
						SIZEOF(a_tyCurrList[1].sRcpNm) , p_udiMax, 1000, 1499, iFilterCtr);
						usiStep := 3;
					3:
						fRecipeFilter(p_sSearch , ADR(a_tyFilterList) , ADR(a_tyCurrList) , SIZEOF(a_tyCurrList[1]) , ADR(a_tyCurrList[1].sRcpNm) ,
						SIZEOF(a_tyCurrList[1].sRcpNm) , p_udiMax, 1500, 1999, iFilterCtr);
						eStatus := Done;

				END_CASE

				eStatus	:= Done;

			END_IF

		MagRcpActLoadRcp:
			IF eStatus = Idle OR eStatus = Busy THEN

				sStatTxt	:= a_sStatText[eStat];

				CASE usiStep OF
					0:	//Get Recipe
						IF p_tyInfoIn.sRcpNm = '' THEN
							bNmEmpty	:= TRUE;
							bNmNotExist	:= TRUE;

							eStatus	:= Done;
						ELSE
							bNmNotExist	:= (fRecipeGetInfo(p_tyInfoIn.sRcpNm , ADR(tyCurrRcp) , ADR(a_tyCurrList) , SIZEOF(a_tyCurrList[1]) , ADR(a_tyCurrList[1].sRcpNm) , SIZEOF(a_tyCurrList[1].sRcpNm) , p_udiMax)) = 0;
							IF bNmNotExist = TRUE THEN
								eStatus	:= Done;
							ELSE
								usiStep	:= 1;
							END_IF
						END_IF

					1:	//Write Into File
						fbFileLoadSingle(bEn := TRUE);

						IF fbFileLoadSingle.udiStatus = 0 THEN
							eStatus			:= Done;
						ELSIF fbFileLoadSingle.udiStatus < 65534 THEN
							eStatus			:= Error;

							IF fbFileLoadSingle.udiStatus = 1900 THEN
								udiStatus	:= 10015;	//File Open Error While Loading Current Recipe
							ELSIF fbFileLoadSingle.udiStatus = 1901 THEN
								udiStatus	:= 10016;	//File Create Error While Loading Current Recipe
							ELSIF fbFileLoadSingle.udiStatus = 1903 THEN
								udiStatus	:= 10017;	//File Write Error While Loading Current Recipe
							ELSIF fbFileLoadSingle.udiStatus = 1904 THEN
								udiStatus	:= 10018;	//File Close Error While Loading Current Recipe
							ELSIF fbFileLoadSingle.udiStatus = 1914 THEN
								udiStatus	:= 10019;	//Directory Does Not Exist While Loading Current Recipe
							ELSE
								udiStatus	:= fbFileLoadSingle.udiStatus;
							END_IF
						END_IF

				END_CASE

			END_IF

		MagRcpActReadCurrRcp:
			IF eStatus = Idle OR eStatus = Busy THEN

				eStatus	:= Busy;

				sStatTxt	:= a_sStatText[eStat];

				fbFileReadSingle(bEn := TRUE);
				IF fbFileReadSingle.udiStatus = 0 THEN
					eStatus	:= Done;

				ELSIF fbFileReadSingle.udiStatus < 65534 THEN
					eStatus		:= Error;

					IF fbFileReadSingle.udiStatus = 1900 THEN
						udiStatus	:= 10020;	//File Open Error While Reading Current Recipe
					ELSIF fbFileReadSingle.udiStatus = 1902 THEN
						udiStatus	:= 10021;	//File Read Error While Reading Current Recipe
					ELSIF fbFileReadSingle.udiStatus = 1904 THEN
						udiStatus	:= 10022;	//File Close Error While Reading Current Recipe
					ELSIF fbFileReadSingle.udiStatus = 1915 THEN
						bFileNotFound	:= TRUE;
						eStatus			:= Done;
					ELSE
						udiStatus	:= fbFileReadSingle.udiStatus;
					END_IF
				END_IF

			END_IF

		MagRcpActWriteCurrRcpParam:
			IF eStatus = Idle OR eStatus = Busy THEN

				sStatTxt	:= a_sStatText[eStat];

				fbFileWriteSingle(bEn := TRUE);

				IF fbFileWriteSingle.udiStatus = 0 THEN
					tyCurrRcp		:= p_tyCurrRcpWr;
					eStatus			:= Done;
				ELSIF fbFileWriteSingle.udiStatus < 65534 THEN
					eStatus			:= Error;

					IF fbFileWriteSingle.udiStatus = 1900 THEN
						udiStatus	:= 10023;	//File Open Error While Writing Current Recipe Parameter
					ELSIF fbFileWriteSingle.udiStatus = 1901 THEN
						udiStatus	:= 10024;	//File Create Error While Writing Current Recipe Parameter
					ELSIF fbFileWriteSingle.udiStatus = 1903 THEN
						udiStatus	:= 10025;	//File Write Error While Writing Current Recipe Parameter
					ELSIF fbFileWriteSingle.udiStatus = 1904 THEN
						udiStatus	:= 10026;	//File Close Error While Writing Current Recipe Parameter
					ELSIF fbFileWriteSingle.udiStatus = 1914 THEN
						udiStatus	:= 10027;	//Directory Does Not Exist While Writing Current Recipe Parameter
					ELSE
						udiStatus	:= fbFileWriteSingle.udiStatus;
					END_IF
				END_IF

			END_IF

		MagRcpActSaveList:
			IF eStatus = Idle OR eStatus = Busy THEN

				eStatus	:= Busy;

				sStatTxt	:= a_sStatText[eStat];

				CASE usiStep OF

					0:
						a_tyListTemp	:= a_tyCurrList;

						fbFileWriteList(bEn := TRUE);

						IF fbFileWriteList.udiStatus = 0 THEN
							eStatus			:= Done;

						ELSIF fbFileWriteList.udiStatus < 65534 THEN
							eStatus			:= Error;

							IF fbFileWriteList.udiStatus = 1900 THEN
								udiStatus	:= 10028;	//File Open Error While Saving List
							ELSIF fbFileWriteList.udiStatus = 1901 THEN
								udiStatus	:= 10029;	//File Create Error While Saving List
							ELSIF fbFileWriteList.udiStatus = 1903 THEN
								udiStatus	:= 10030;	//File Write Error While Saving List
							ELSIF fbFileWriteList.udiStatus = 1904 THEN
								udiStatus	:= 10031;	//File Close Error While Saving List
							ELSIF fbFileWriteList.udiStatus = 1914 THEN
								udiStatus	:= 10032;	//Directory Does Not Exist While Saving List
							ELSE
								udiStatus	:= fbFileWriteList.udiStatus;
							END_IF
						END_IF

				END_CASE

			END_IF

		MagRcpActSort:
			IF eStatus = Idle OR eStatus = Busy THEN

				sStatTxt	:= a_sStatText[eStat];

				CASE usiStep OF

					0:

						FOR udi := 1 TO c_udiMagRcpMax DO
							IF p_sSearch <> '' THEN
								IF a_tyFilterList[udi].sRcpNm = '' THEN
									usiStep := 1;
									EXIT;
								ELSIF udi = c_udiMagRcpMax THEN
									iTotalRcp := UDINT_TO_INT(c_udiMagRcpMax);
									usiStep := 1;
									EXIT;
								ELSE
									iTotalRcp := iTotalRcp +1;
								END_IF
							ELSE
								IF a_tyCurrList[udi].sRcpNm = '' THEN
									usiStep := 1;
									EXIT;
								ELSIF udi = c_udiMagRcpMax THEN
									iTotalRcp := UDINT_TO_INT(c_udiMagRcpMax);
									usiStep := 1;
									EXIT;
								ELSE
									iTotalRcp := iTotalRcp +1;
								END_IF
							END_IF
						END_FOR

					1:
						IF p_sSearch <> '' THEN
							memcpy(ADR(a_tySortList),ADR(a_tyFilterList), SIZEOF(a_tyFilterList));
						ELSE
							memcpy(ADR(a_tySortList),ADR(a_tyCurrList), SIZEOF(a_tyCurrList));
						END_IF

						iSortCurrentOuterCntr	:= 0;
						iSortCurrentInnerCntr	:= 1 ;

						udiSortCurrenTotalCntr	:= 0;

						usiStep := 2;

					2:

						IF iSortCurrentOuterCntr < iTotalRcp THEN

							FOR iSortCurrentInnerCntr:= iSortCurrentOuterCntr+1 TO iTotalRcp-1 DO

								IF fRecipeNmCompare(ADR(a_tySortList[iSortCurrentOuterCntr+1].sRcpNm),ADR(a_tySortList[iSortCurrentInnerCntr+1].sRcpNm),SIZEOF(a_tySortList[1].sRcpNm),ADR(sDebug)) THEN

									memcpy(ADR(tyTempRecipe), ADR(a_tySortList[iSortCurrentOuterCntr+1]), SIZEOF(a_tySortList[1]));
									memcpy(ADR(a_tySortList[iSortCurrentOuterCntr+1]), ADR(a_tySortList[iSortCurrentInnerCntr+1]), SIZEOF(a_tySortList[1]));
									memcpy(ADR(a_tySortList[iSortCurrentInnerCntr+1]), ADR(tyTempRecipe), SIZEOF(a_tySortList[1]));

								END_IF

								udiSortCurrenTotalCntr	:= udiSortCurrenTotalCntr + 1;

							END_FOR

							iSortCurrentOuterCntr	:= iSortCurrentOuterCntr + 1;

						ELSE
							usiStep := 3;
						END_IF

					3:
						eStatus	:= Done;

				END_CASE

			END_IF

	END_CASE

END_ACTION
```

#### Cyclic.st
```iecst
(** 2019-03-29 **)
PROGRAM _CYCLIC

	IF bInitDone = FALSE THEN
		bInitDone	:= TRUE;

		Act_InitLocal;
		Act_InitGlobal;

	ELSIF bInitialDone = FALSE THEN
		IF p_bNtSettingsLoadDone = TRUE THEN
			bInitialDone	:= TRUE;

			Act_Initial;
		END_IF

	ELSE

		Act_RstErr;
		Act_LinkAction;
		Act_Action;
		Act_LinkEn;

		IF p_bPrep = TRUE AND p_bDis = FALSE THEN
			Act_Link;
			Act_Main;
		ELSE
			IF eStat <> MagRcpActIdle THEN
				eStatus	:= Done;
			ELSE
				eStatus	:= Idle;
			END_IF
		END_IF

		Act_Alarm;

	END_IF

END_PROGRAM
```

#### Init.st
```iecst
(** 2019-05-04 **)
PROGRAM _INIT

	(* Always Change If Project Change *)

	//Pass Address To Global Address For External Use
	//Action, State & Status
	p_MagRcpStat	:= ADR(eStat);
	p_MagRcpStatus	:= ADR(eStatus);
	p_MagRcpStatTxt	:= ADR(sStatTxt);

	//Alarm
	p_MagRcpAlmData	:= ADR(tyAlmData);

	//Output
	p_MagRcpNmExist			:= ADR(bNmExist);
	p_MagRcpNmNotExist		:= ADR(bNmNotExist);
	p_MagRcpNmEmpty			:= ADR(bNmEmpty);
	p_MagRcpListFull		:= ADR(bListFull);
	p_MagRcpCurrList		:= ADR(a_tyCurrList);
	p_MagRcpFilterList		:= ADR(a_tyFilterList);
	p_MagRcpSortedList		:= ADR(a_tySortList);
	p_MagRcpInfoOut			:= ADR(tyInfoOut);
	p_MagRcpFileNotFound	:= ADR(bFileNotFound);

	p_MagRcpCurrRcp					:= ADR(tyCurrRcp);
	p_MagRcpCurrRcpNm				:= ADR(tyCurrRcp.sRcpNm);
	p_MagRcpCurrRcpTtlSlt			:= ADR(tyCurrRcp.diTtlSlt);
	p_MagRcpCurrRcpSltToSlt			:= ADR(tyCurrRcp.diSltToSltInUM);
	p_MagRcpCurrRcpMag1Slt1Pos		:= ADR(tyCurrRcp.diMag1Slt1PosInUM);
	p_MagRcpCurrRcpMag2Slt1Pos		:= ADR(tyCurrRcp.diMag2Slt1PosInUM);
	p_MagRcpCurrRcpMag3Slt1Pos		:= ADR(tyCurrRcp.diMag3Slt1PosInUM);
	p_MagRcpCurrRcpMag1TravPos		:= ADR(tyCurrRcp.diMag1TravPosInUM);
	p_MagRcpCurrRcpMag2TravPos		:= ADR(tyCurrRcp.diMag2TravPosInUM);
	p_MagRcpCurrRcpMag3TravPos		:= ADR(tyCurrRcp.diMag3TravPosInUM);
	p_MagRcpCurrRcpDisplayInfo		:= ADR(tyCurrRcp.sDisplayInfo);
	p_MagRcpCurrRcpLastModified		:= ADR(tyCurrRcp.dtLastModified);
	p_MagRcpCurrRcpMagMaxBrdWidth	:= ADR(tyCurrRcp.diMagMaxBrdWidth);
	p_MagRcpCurrRcpMagModel			:= ADR(tyCurrRcp.usiMagModel);
	p_MagRcpCurrRcpSBarDisabled		:= ADR(tyCurrRcp.bSafetyBarDisabled);
	p_MagRcpCurrRcpMagHeightChkEn	:= ADR(tyCurrRcp.bMagHeightChkEn);
	(* Always Change If Project Change *)

END_PROGRAM
```

### McParam.typ - Change By Project
```iecst
(*2019-05-04*)
(**)
(*Action*)

TYPE
	eMcParamAction :
		(
		McParamActIdle,
		McParamActCreateDir,
		McParamActRead,
		McParamActWrite
		);
	tyMcParam : 	STRUCT
		a_bLFOnline : ARRAY[1..c_diLFClntNum]OF BOOL;
		a_sLFIPAddr : ARRAY[1..c_diLFClntNum]OF STRING[15];
		sMcNm : STRING[30] := 'Triple Magazine Line Unloader';
		uiSSaverTmInSec : UINT := 1800;
		bSSaverEn : BOOL := FALSE;
		usiDefaultMcMod : USINT := 0;
		diAWPusherAtHmPosInUM : DINT := 0;
		diWidthAtHmPosInUM : DINT := 0;
		diConvInitTmInMS : DINT := 6000;
		diTranInErrDlyTmInMS : DINT := 12000;
		diMag1ConvRunTmOutInMS : DINT := 20000;
		diMag2ConvRunTmOutInMS : DINT := 20000;
		diMag3ConvRunTmOutInMS : DINT := 20000;
		diOvenMaxBffr : DINT := 1;
		diTravPosA : DINT;
		diTravPosB : DINT;
		diLifterPosA : DINT;
		diLifterPosB : DINT;
		bAWPusherDis : BOOL := FALSE;
		bAWDis : BOOL := FALSE;
		bMnlAccDat : BOOL := FALSE;
		bAutoStepEn : BOOL := FALSE;
		bVSMEMAEn : BOOL := TRUE;
		bChgParamEn : BOOL := TRUE;
		bHermesRmtEn : BOOL := FALSE;
		bHermesSvyEn : BOOL := FALSE;
		bHermesScannerEn : BOOL;
		bGapBwtnBrdEn : BOOL := FALSE;
		bLongBrdEn : BOOL := FALSE;
		bOvenEn : BOOL := FALSE;
		bExtdOvenEn : BOOL := FALSE;
		bInShutterDis : BOOL := FALSE;
		bStopperADis : BOOL := FALSE;
		bStopperBDis : BOOL := FALSE;
		bLFEn : BOOL := FALSE;
		bLCSLFEn : BOOL := FALSE;
		bLCSReqRcpEn : BOOL := FALSE;
		bLCSManageRcpEn : BOOL := FALSE;
		bLCSLiveDatEn : BOOL := FALSE;
		bLFLeaderMc : BOOL := FALSE;
		bSectionLeader : BOOL := FALSE;
		bUSWidthChkEn : BOOL := FALSE;
		diWidthOffsetInUM : DINT := 0;
		diLFMcIdxBeforeOven : DINT := 1;
		diLFMcIdxAfterOven : DINT := 1;
		diLFMcIdxBeforeOven2 : DINT := 1;
		diLFMcIdxAfterOven2 : DINT := 1;
		usiLang : USINT := 0;
		tyLftSenAntiGapDly : tyAntiGapDly := (diSigOnTm:=0,diSigOffTm:=100);
		tyMidSenAntiGapDly : tyAntiGapDly := (diSigOnTm:=0,diSigOffTm:=0);
		tyRgtSenAntiGapDly : tyAntiGapDly := (diSigOnTm:=0,diSigOffTm:=500);
		tyClrSenAntiGapDly : tyAntiGapDly := (diSigOnTm:=0,diSigOffTm:=500);
		eUSCommA : eMcSetCommMod := McSetCommModSMEMA;
		tyUSCommASMEMA : tySMEMAParam := (eSelection:=SMEMASelIPC9851,bStatSigSetGd:=FALSE);
		eUSCommB : eMcSetCommMod := McSetCommModSMEMA;
		bAutoLogoutEn : BOOL := FALSE;
		diAutoLogoutTmInSec : DINT := 60000;
		sIPAddr : STRING[15] := '192.168.0.10';
		sSubnetMask : STRING[15] := '255.255.255.0';
		eNetworkMod : eNetworkConfigMod := SetIPManually;
		tyUSCommBSMEMA : tySMEMAParam := (eSelection:=SMEMASelIPC9851,bStatSigSetGd:=FALSE);
		diMagAutoDetectSenTmInMS : DINT := 2000;
		bAGVComEn : BOOL := FALSE;
		tyMagConvEntrySenAntiGapDly : tyAntiGapDly := (diSigOnTm:=100,diSigOffTm:=100);
		tyMagConvPresentSenAntiGapDly : tyAntiGapDly := (diSigOnTm:=100,diSigOffTm:=100);
		bLFSeqStayActive : BOOL := FALSE;
		bMagAWDis : BOOL := FALSE;
		bMagSafetyBarDis : BOOL := FALSE;
		diMag1WidthAtHmPosInUM : DINT;
		diMag2WidthAtHmPosInUM : DINT;
		diMag3WidthAtHmPosInUM : DINT;
		bLFBuzMute : BOOL := FALSE;
		eAGVComProtocol : eMcAGVCommProtocol := McSetAGVCommOPCUA;
		eMagExMode : eMcMagExchangeMode := McSetMagXcAutoManMode;
		bAIVSizeDisabled : BOOL := FALSE;
		diTravInletFixtoFixPos : DINT := 0;
		bDisableFMWarning : BOOL := TRUE;
		tyLineAInletSenAntiGapDly : tyAntiGapDly := (diSigOnTm:=0,diSigOffTm:=0);
		tyLineBInletSenAntiGapDly : tyAntiGapDly := (diSigOnTm:=0,diSigOffTm:=0);
		tyUSWidthChkSenAntiGapDly : tyAntiGapDly := (diSigOnTm:=0,diSigOffTm:=0);
		bDBAOnWOAlign : BOOL := FALSE;
		tyInMagConvEntAntiGapDly : tyAntiGapDly := (diSigOnTm:=0,diSigOffTm:=0);
		tyInMagConvMidAntiGapDly : tyAntiGapDly := (diSigOnTm:=0,diSigOffTm:=0);
		tyInMagConvExtAntiGapDly : tyAntiGapDly := (diSigOnTm:=0,diSigOffTm:=0);
		tyOutMagConvEntAntiGapDly : tyAntiGapDly := (diSigOnTm:=1500,diSigOffTm:=1500);
		tyOutMagConvMidAntiGapDly : tyAntiGapDly := (diSigOnTm:=0,diSigOffTm:=0);
		tyOutMagConvExtAntiGapDly : tyAntiGapDly := (diSigOnTm:=0,diSigOffTm:=1200);
		tyInMagConv2EntAntiGapDly : tyAntiGapDly := (diSigOnTm:=0,diSigOffTm:=0);
		tyInMagConv2MidAntiGapDly : tyAntiGapDly := (diSigOnTm:=0,diSigOffTm:=0);
		tyInMagConv2ExtAntiGapDly : tyAntiGapDly := (diSigOnTm:=0,diSigOffTm:=0);
		tyOutMagConv2EntAntiGapDly : tyAntiGapDly := (diSigOnTm:=1500,diSigOffTm:=1500);
		tyOutMagConv2MidAntiGapDly : tyAntiGapDly := (diSigOnTm:=0,diSigOffTm:=0);
		tyOutMagConv2ExtAntiGapDly : tyAntiGapDly := (diSigOnTm:=0,diSigOffTm:=1200);
		diInMagConvRunTmOutInMS : DINT := 20000;
		diOutMagConvRunTmOutInMS : DINT := 20000;
		diLifterMagConvRunTmOutInMS : DINT := 20000;
		diInMagConv2RunTmOutInMS : DINT := 20000;
		diOutMagConv2RunTmOutInMS : DINT := 20000;
		diLifterMagConv2RunTmOutInMS : DINT := 20000;
		diLifterTopPos : DINT := 0;
		diLifterBtmPos : DINT := 0;
		diLifterTopPos2 : DINT := 0;
		diLifterBtmPos2 : DINT := 0;
		diTCPSvrPort : DINT := 7171;
		bMagWidthChkDis : BOOL := TRUE;
		diMag1WidthChkDetDist : DINT := 2000;
		diMag2WidthChkDetDist : DINT := 2000;
		diMag3WidthChkDetDist : DINT := 2000;
		bTopScannerEn : BOOL;
		bBtmScannerEn : BOOL;
		sTopScanIPAddr : STRING[15] := '192.168.2.100';
		uiTopScanSvrPort : UINT := 51236;
		sBtmScanIPAddr : STRING[15] := '192.168.2.101';
		uiBtmScanSvrPort : UINT := 51237;
		bOpConEn : BOOL;
		sOpConIPAddr : STRING[15] := '192.168.0.102';
		uiOpConSvrPort : UINT := 51238;
		tyOpConParam : tyLocationParamData := (uiLineNo:=1,uiStatNo:=1,uiStatIdx:=1,uiFuNo:=1,uiWorkPos:=1,uiToolPos:=1,uiProcessNo:=1,sApplication:='IPC');
		bSiemensPrep : BOOL;
		bInStopperDis : BOOL;
		diInletStopperExtDelayTmInMS : DINT;
		diMESResponseTOTmInMS : DINT;
		bMESEn : BOOL;
		bSwitchingProdType : BOOL;
		bAutoRcpDisable : BOOL;
		bBatchIDChgOverCmp : BOOL;
		bIgnoreTopClearance : BOOL;
		bIgnoreBtmClearance : BOOL;
		bIgnoreThickness : BOOL;
		bDMCScannerEn : BOOL := FALSE;
		diDMCScanTOErrInMs : DINT;
		tyOptBtnPos : tyBtnPos := (ePos1:=eMagUnload,ePos2:=eNA,ePos3:=eNA);
		sHMIIPAddr : STRING[15] := '192.168.0.11';
		sDefaultGateWay : STRING[15] := '0.0.0.0';
	END_STRUCT;
	tyMcParamGen : 	STRUCT
		In : tyMcParamIn1;
		Out : tyMcParamOut1;
	END_STRUCT;
	tyMcParamIn1 : 	STRUCT
		eAct : eMcParamAction;
		udiRstErr : UDINT;
		tyMcParmWr : tyMcParam;
		sProgNm : STRING[15];
	END_STRUCT;
	tyMcParamOut1 : 	STRUCT
		eStat : eMcParamAction;
		eStatus : eFBStatus;
		sStatTxt : STRING[200];
		tyAlmData : tyAlmDat;
		bFileNotFound : BOOL;
	END_STRUCT;
END_TYPE

(**)

TYPE
	tyAntiGapDly : 	STRUCT
		diSigOnTm : DINT;
		diSigOffTm : DINT;
	END_STRUCT;
	eMcSetCommMod :
		(
		McSetCommModSMEMA,
		McSetCommModHermes
		);
	eMcAGVCommProtocol :
		(
		McSetAGVCommOPCUA,
		McSetAGVCommHardIO,
		McSetAGVCommDisabled,
		McSetAGVTCPEnableTCP,
		McSetAGVTCPDisableTCP
		);
	eMcMagExchangeMode :
		(
		McSetMagXcAutoManMode,
		McSetMagXcAutoMode,
		McSetMagXcManMode
		);
END_TYPE

(**)

TYPE
	tyBtnPos : 	STRUCT
		ePos1 : eOptBtn := eNA;
		ePos2 : eOptBtn := eRlsNewMagazine1;
		ePos3 : eOptBtn := eRlsNewMagazine2;
		ePos4 : eOptBtn := eRlsNewMagazine3;
		ePos5 : eOptBtn := eRlsNewMagazine3;
		ePos6 : eOptBtn := eRlsNewMagazine3;
		ePos7 : eOptBtn := eRlsNewMagazine3;
	END_STRUCT;
	eOptBtn :
		(
		eNA := 0,
		eMagUnload := 1,
		eRlsNewMagazine1 := 2,
		eRlsNewMagazine2 := 3,
		eRlsNewMagazine3 := 4
		);
END_TYPE
```

### McParam.var - Change By Project
```iecst
(*2019-04-17*)
VAR
	g_tyMcParamCurr : tyMcParam;
	g_tyMcParamOut : tyMcParamOut1;
END_VAR
(**)
```

### Program Logical/McParam/McParam (IEC, version 1.00.0)

#### Act_InputConfig.st - Change By Project
```iecst
ACTION Act_InputConfig:

	tylocalMcParam.In.udiRstErr 	:= g_tyRstErrOut.udiRstErr;
	tylocalMcParam.In.tyMcParmWr	:= g_tyUIOut.tyMcParamWr;
	tylocalMcParam.In.sProgNm		:= g_tyNtParamCurr.sMcParamProgNm;

	IF g_tyStartUp.bRun THEN
		tylocalMcParam.In.eAct  := g_tyStartUp.eMcParamAct;
	ELSIF g_tySvyHermes.bWriteConfig THEN
		tylocalMcParam.In.eAct  := g_tySvyHermes.eMcParamAct;
	ELSIF g_tyRmtHermes.bWriteConfig THEN
		tylocalMcParam.In.eAct  := g_tyRmtHermes.eMcParamAct;
	ELSE
		tylocalMcParam.In.eAct	:= g_tyUIOut.eMnlAct.eMcParamAct;
	END_IF

END_ACTION
```

#### Act_OutputConfig.st - Change By Project
```iecst
ACTION Act_OutputConfig:

	g_tyMcParamCurr := tyMcParamCurr;
	g_tyMcParamOut  := tylocalMcParam.Out;

END_ACTION
```

#### Cyclic.st - Do Not Change!!!
```iecst
(** 2019-03-29 **)
PROGRAM _CYCLIC

	IF bInitialDone = FALSE THEN
		IF g_tyStartUp.bNtSettingsLoadDone = TRUE THEN
			bInitialDone	:= TRUE;
			Act_Initial;
		END_IF

	ELSE

		Act_InputConfig;
		Act_Link;
		Act_Main;
		Act_OutputConfig;
		Act_Alarm;

	END_IF

END_PROGRAM
```

#### Act_Initial.st - Do Not Change!!!
```iecst
(** 2019-01-15 **)
ACTION Act_Initial:

	//Initial
	sStatTxt	:= a_sStatText[tylocalMcParam.Out.eStat];

	fbDirCreate1.sDevice	:= 'F';
	fbDirCreate1.sDirName	:= 'User';
	fbDirCreate1(bEn := FALSE);

	fbDirCreate2.sDevice	:= 'User';
	fbDirCreate2.sDirName	:= 'MachineParameter';
	fbDirCreate2(bEn := FALSE);

	fbFileRead1.sDevice			:= 'McParam';
	fbFileRead1.sFile			:= g_tyNtParamCurr.sMcParamFileNm;
	fbFileRead1.udiOffset		:= 0;
	fbFileRead1.p_Dest			:= ADR(tyMcParamCurr);
	fbFileRead1.udiLen			:= SIZEOF(tyMcParamCurr);
	fbFileRead1(bEn := FALSE);

	fbFileWrite1.sDevice		:= 'McParam';
	fbFileWrite1.sFile			:= g_tyNtParamCurr.sMcParamFileNm;
	fbFileWrite1.udiOffset		:= 0;
	fbFileWrite1.p_Src			:= ADR(tylocalMcParam.In.tyMcParmWr);
	fbFileWrite1.udiLen			:= SIZEOF(tylocalMcParam.In.tyMcParmWr);
	fbFileWrite1.udiOption		:= 0;
	fbFileWrite1(bEn := FALSE);

	fbFileWrite2.sDevice		:= 'McParam';
	fbFileWrite2.sFile			:= g_tyNtParamCurr.sMcParamFileNm;
	fbFileWrite2.udiOffset		:= 0;
	fbFileWrite2.p_Src			:= ADR(tyMcParamTemp);
	fbFileWrite2.udiLen			:= SIZEOF(tyMcParamTemp);
	fbFileWrite2.udiOption		:= 0;
	fbFileWrite2(bEn := FALSE);

	sVNCAddrNodeID := '54267'; // HMI VNC's IP Address Node ID
	sHMIAddrNodeID := '54248'; // HMI Network's IP Address Node ID
	sObjIDNodeID := '54159'; // HMI MethodSet's Node ID
	sSaveCfgNodeID := '54322'; // HMI Save Method's Node ID
	sLoadCfgNodeID := '54321'; // HMI Load Method's Node ID

	uiNSIdx := 4;
	fbConnectOPCUA.tyOPCUAParam.sPort := '4841';
	fbConnectOPCUA(bEn := FALSE);
	fbReadGetNodeHdlList.usiNSIdx := uiNSIdx;
	fbReadGetNodeHdlList.uiTagNmCnt := 2;
	fbReadGetNodeHdlList.a_sServerTagNm[0] := sVNCAddrNodeID;
	fbReadGetNodeHdlList.a_sServerTagNm[1] := sHMIAddrNodeID;
	fbReadGetNodeHdlList(bEn := FALSE);
	fbReadList.uiTagNmCnt := 2;
	fbReadList(bEn := FALSE);

	fbWriteGetNodeHdlList.usiNSIdx := uiNSIdx;
	fbWriteGetNodeHdlList.uiTagNmCnt := 2;
	fbWriteGetNodeHdlList.a_sServerTagNm[0] := sVNCAddrNodeID;
	fbWriteGetNodeHdlList.a_sServerTagNm[1] := sHMIAddrNodeID;
	fbWriteGetNodeHdlList(bEn := FALSE);
	fbWriteList.uiTagNmCnt := 2;
	fbWriteList(bEn := FALSE);

	fbSaveCfgMethodGetHdl.uiNSIdx := uiNSIdx;
	fbSaveCfgMethodGetHdl.sObjectIdentifier := sObjIDNodeID;
	fbSaveCfgMethodGetHdl.sMethodIdentifier := sSaveCfgNodeID;
	fbSaveCfgMethodGetHdl(bEn := FALSE);
	fbSaveCfgMethodCall(bEn := FALSE);

	fbLoadCfgMethodGetHdl.uiNSIdx := uiNSIdx;
	fbLoadCfgMethodGetHdl.sObjectIdentifier := sObjIDNodeID;
	fbLoadCfgMethodGetHdl.sMethodIdentifier := sLoadCfgNodeID;
	fbLoadCfgMethodGetHdl(bEn := FALSE);
	fbLoadCfgMethodCall(bEn := FALSE);

	fbDisconnectOPCUA(bEn := FALSE);
END_ACTION
```

#### Act_Link.st - Change By Project
```iecst
(** 2021-08-08 **)
ACTION Act_Link:

	IF tyMcParamCurr.eAGVComProtocol = McSetAGVCommOPCUA
		OR tyMcParamCurr.eAGVComProtocol = McSetAGVCommHardIO
		OR tyMcParamCurr.eAGVComProtocol = McSetAGVTCPEnableTCP
		THEN
		IF tyMcParamCurr.eMagExMode = McSetMagXcAutoManMode
			OR tyMcParamCurr.eMagExMode = McSetMagXcAutoMode
			THEN
			tyMcParamCurr.bAGVComEn := TRUE;
		ELSE
			tyMcParamCurr.bAGVComEn := FALSE;
		END_IF
	ELSIF tyMcParamCurr.eAGVComProtocol = McSetAGVCommDisabled OR tyMcParamCurr.eAGVComProtocol = McSetAGVTCPDisableTCP THEN
		tyMcParamCurr.bAGVComEn := FALSE;
	END_IF

	//new for Hermes 1.3
		//Changed
	IF g_tyRmtHermes.bWriteConfig OR g_tySvyHermes.bWriteConfig THEN
		tylocalMcParam.In.tyMcParmWr.sMcNm := g_tySvyHermes.tyHermesConfigurationWr.tySvyParam.sMachineId;//p_tyHermesConfigurationWr.tySvyParam.sMachineId;
	END_IF

	//Control AutoRcp
	IF NOT(g_tyNtParamCurr.bAutoRcpPrep) THEN
		tyMcParamCurr.bAutoRcpDisable := TRUE;
	ELSE
		//auto rcp prep
		CASE g_tyNtParamCurr.eAutoRcpPrecededBy OF
			PrecededBySelf:
				IF tyMcParamCurr.eUSCommA <> McSetCommModHermes AND ( NOT(g_tyNtParamCurr.bProjLaneBPrep) OR (g_tyNtParamCurr.bProjLaneBPrep AND tyMcParamCurr.eUSCommB <> McSetCommModHermes)) THEN
					tyMcParamCurr.bAutoRcpDisable := TRUE;
				ELSE
					tyMcParamCurr.bAutoRcpDisable := FALSE;
				END_IF
			PrecededByF1:
				tyMcParamCurr.bAutoRcpDisable := FALSE; //for LCS
			ELSE
				tyMcParamCurr.bAutoRcpDisable := FALSE;
		END_CASE
	END_IF

	//Disable MES on SMEMA mode
	IF g_tyNtParamCurr.eCustomerReq = Siemens AND tyMcParamCurr.eUSCommA <> McSetCommModHermes  AND ( NOT(g_tyNtParamCurr.bProjLaneBPrep) OR (g_tyNtParamCurr.bProjLaneBPrep AND tyMcParamCurr.eUSCommB <> McSetCommModHermes)) THEN
		tyMcParamCurr.bMESEn := TRUE;
		tyMcParamCurr.bHermesSvyEn := FALSE;
	END_IF

	IF g_tyStartUp.bRun = FALSE THEN

		CASE usiChkIpAddrStep OF

			0:
				//Connect HMI OPCUA Server
				fbConnectOPCUA.tyOPCUAParam.sIPAddr	:= tyMcParamCurr.sHMIIPAddr;
				fbConnectOPCUA(bEn := TRUE);

				IF fbConnectOPCUA.udiStatus = 0 THEN
					dwConnectionHdl	:= fbConnectOPCUA.dwConnectionHdl;
					fbConnectOPCUA(bEn := FALSE);

					bConnected := TRUE;

					usiChkIpAddrStep	:= 1;
				ELSIF fbConnectOPCUA.udiStatus < 65534 THEN
					fbConnectOPCUA(bEn := FALSE);

					bConnected := FALSE;
					usiChkIpAddrStep := 0;
				END_IF

			1:
				//Node Handle List Read
				fbReadGetNodeHdlList.dwConnectionHdl := dwConnectionHdl;
				fbReadGetNodeHdlList(bEn := TRUE);

				IF fbReadGetNodeHdlList.udiStatus = 0 THEN
					tyReadHdls.a_dwHdls := fbReadGetNodeHdlList.a_dwNodeHdlList;
					fbReadGetNodeHdlList(bEn := FALSE);

					usiChkIpAddrStep := 2;
				ELSIF fbReadGetNodeHdlList.udiStatus < 65534 THEN
					fbReadGetNodeHdlList(bEn := FALSE);

					usiChkIpAddrStep := 9;
				END_IF

			2:
				//Read List
				fbReadList.dwConnectionHdl := dwConnectionHdl;
				fbReadList.a_dwNodeHdlList := tyReadHdls.a_dwHdls;

				fbReadList.a_sClientTagNm[0] := '::McParam:sVNCIPAddr';
				fbReadList.a_sClientTagNm[1] := '::McParam:sHMIIPAddr';
				fbReadList(bEn := TRUE);

				IF fbReadList.udiStatus = 0 THEN
					fbReadList(bEn := FALSE);

					IF g_tyHWInfo.sIPAddr <> sVNCIPAddr OR g_tyUIOut.bUpdtHMIIPAddr  THEN

						usiChkIpAddrStep := 3;
					END_IF

				ELSIF fbReadList.udiStatus < 65534 THEN
					fbReadList(bEn := FALSE);

					usiChkIpAddrStep := 9;
				END_IF

			3:
				//Node Handle List Write
				eStatus := Busy;

				fbWriteGetNodeHdlList.dwConnectionHdl := dwConnectionHdl;
				fbWriteGetNodeHdlList(bEn := TRUE);

				IF fbWriteGetNodeHdlList.udiStatus = 0 THEN
					tyWriteHdls.a_dwHdls := fbWriteGetNodeHdlList.a_dwNodeHdlList;
					fbWriteGetNodeHdlList(bEn := FALSE);

					usiChkIpAddrStep := 4;
				ELSIF fbWriteGetNodeHdlList.udiStatus < 65534 THEN
					fbWriteGetNodeHdlList(bEn := FALSE);

					usiChkIpAddrStep := 9;
				END_IF

			4:
				//Write List
				fbWriteList.dwConnectionHdl := dwConnectionHdl;

				fbWriteList.a_dwNodeHdlList := tyWriteHdls.a_dwHdls;

				sVNCIPAddr	:= g_tyHWInfo.sIPAddr;

				IF LEN(g_tyUIOut.sSetHMIIPAddr) > 0 THEN
					sHMIIPAddr	:= g_tyUIOut.sSetHMIIPAddr;
				ELSE
					sHMIIPAddr	:= tyMcParamCurr.sHMIIPAddr;
				END_IF

				fbWriteList.a_sClientTagNm[0] := '::McParam:sVNCIPAddr';
				fbWriteList.a_sClientTagNm[1] := '::McParam:sHMIIPAddr';
				fbWriteList(bEn := TRUE);

				IF fbWriteList.udiStatus = 0 THEN
					fbWriteList(bEn := FALSE);

					usiChkIpAddrStep := 5;
				ELSIF fbWriteList.udiStatus < 65534 THEN
					fbWriteList(bEn := FALSE);

					usiChkIpAddrStep := 9;
				END_IF

			5:
				//Method Get Handle (Save Configuration)
				fbSaveCfgMethodGetHdl.dwConnectionHdl := dwConnectionHdl;
				fbSaveCfgMethodGetHdl(bEn := TRUE);

				IF fbSaveCfgMethodGetHdl.udiStatus = 0 THEN
					dwMethodHdl	:= fbSaveCfgMethodGetHdl.dwMethodHdl;
					fbSaveCfgMethodGetHdl(bEn := FALSE);

					usiChkIpAddrStep := 6;
				ELSIF fbSaveCfgMethodGetHdl.udiStatus < 65534 THEN
					fbSaveCfgMethodGetHdl(bEn := FALSE);

					usiChkIpAddrStep := 9;
				END_IF

			6:
				//Method Call (Save Configuration)
				fbSaveCfgMethodCall.dwConnectionHdl		:= dwConnectionHdl;
				fbSaveCfgMethodCall.dwMethodHdl			:= dwMethodHdl;

				fbSaveCfgMethodCall(bEn	:= TRUE);

				IF fbSaveCfgMethodCall.udiStatus = 0 THEN
					fbSaveCfgMethodCall	(bEn := FALSE);

					usiChkIpAddrStep	:= 7;
				ELSIF fbSaveCfgMethodCall.udiStatus	< 65534 THEN
					fbSaveCfgMethodCall(bEn := FALSE);

					usiChkIpAddrStep	:= 9;
				END_IF

			7:
				//Method Get Handle (Load Configuration)
				fbLoadCfgMethodGetHdl.dwConnectionHdl		:= dwConnectionHdl;
				fbLoadCfgMethodGetHdl(bEn := TRUE);

				IF fbLoadCfgMethodGetHdl.udiStatus = 0 THEN
					dwMethodHdl	:= fbLoadCfgMethodGetHdl.dwMethodHdl;
					fbLoadCfgMethodGetHdl(bEn := FALSE);

					usiChkIpAddrStep := 8;
				ELSIF fbLoadCfgMethodGetHdl.udiStatus < 65534 THEN
					fbLoadCfgMethodGetHdl(bEn := FALSE);
					dwMethodHdl	:= 0;

					usiChkIpAddrStep := 9;
				END_IF

			8:
				//Method Call (Load Configuration)
				fbLoadCfgMethodCall.dwConnectionHdl			:= dwConnectionHdl;
				fbLoadCfgMethodCall.dwMethodHdl				:= dwMethodHdl;
				fbLoadCfgMethodCall(bEn := TRUE);

				IF fbLoadCfgMethodCall.udiStatus = 0 THEN
					fbLoadCfgMethodCall(bEn := FALSE);

					usiChkIpAddrStep	:= 9;
				ELSIF fbLoadCfgMethodCall.udiStatus < 65534 THEN
					fbLoadCfgMethodCall(bEn := FALSE);

					usiChkIpAddrStep := 9;
				END_IF

			9:
				//Disconnect
				fbDisconnectOPCUA.dwConnectionHdl		:= dwConnectionHdl;
				fbDisconnectOPCUA(bEn := TRUE);

				IF fbDisconnectOPCUA.udiStatus = 0 THEN
					fbDisconnectOPCUA(bEn := FALSE);
					dwConnectionHdl	:= 0;
					dwMethodHdl		:= 0;
					eStatus := Done;

					usiChkIpAddrStep	:=0;

				ELSIF fbDisconnectOPCUA.udiStatus < 65534 THEN
					fbDisconnectOPCUA(bEn := FALSE);
					dwConnectionHdl := 0;
					bConnected := FALSE;
					udiStatus			:= 10013; //Failed to Call Load Configuration Method

					usiChkIpAddrStep := 0;
				END_IF

		END_CASE

		IF bConnected = FALSE THEN
			udiStatus := 10010;

			//eStatus := Error;
			IF dwConnectionHdl = 0 THEN

				IF LEN(sHMIIPAddr) > 0 THEN
					tyMcParamCurr.sHMIIPAddr := sHMIIPAddr;
				ELSIF LEN(g_tyUIOut.sSetHMIIPAddr) > 0 THEN
					tyMcParamCurr.sHMIIPAddr := g_tyUIOut.sSetHMIIPAddr;
				END_IF

			ELSE
				dwConnectionHdl := 0;
			END_IF

		ELSIF bConnected = TRUE AND udiStatus = 10010 THEN
			bRstErr := TRUE;
		END_IF
	END_IF
END_ACTION
```

#### Act_Main.st - Do Not Change!!!
```iecst
(** 2019-01-10 **)
ACTION Act_Main:
	IF tylocalMcParam.Out.eStatus = Idle THEN
		tylocalMcParam.Out.eStat	:= tylocalMcParam.In.eAct;
	END_IF

	//Main
	CASE tylocalMcParam.Out.eStat OF

		McParamActIdle:
			IF tylocalMcParam.Out.eStatus <> Idle THEN	//Reset Data
				//Private
				fbDirCreate1(bEn := FALSE);
				fbDirCreate2(bEn := FALSE);
				fbFileRead1(bEn := FALSE);
				fbFileWrite1(bEn := FALSE);
				fbFileWrite2(bEn := FALSE);
				usiStep	:= 0;

				bFileNotFound	:= FALSE;

				sStatTxt	:= a_sStatText[tylocalMcParam.Out.eStat];

			END_IF

			tylocalMcParam.Out.eStatus	:= Idle;

		McParamActCreateDir:
			IF tylocalMcParam.Out.eStatus = Idle OR tylocalMcParam.Out.eStatus = Busy THEN

				tylocalMcParam.Out.eStatus	:= Busy;

				sStatTxt	:= a_sStatText[tylocalMcParam.Out.eStat];

				CASE usiStep OF
					0:
						fbDirCreate1(bEn := TRUE);
						IF fbDirCreate1.udiStatus = 0 THEN
							usiStep	:= 1;
						ELSIF fbDirCreate1.udiStatus < 65534 THEN
							tylocalMcParam.Out.eStatus		:= Error;

							IF fbDirCreate1.udiStatus = 1908 THEN
								udiStatus	:= 10000;	//Create User Directory Error
							ELSE
								udiStatus	:= fbDirCreate1.udiStatus;
							END_IF
						END_IF

					1:
						fbDirCreate2(bEn := TRUE);
						IF fbDirCreate2.udiStatus = 0 THEN
							tylocalMcParam.Out.eStatus	:= Done;
						ELSIF fbDirCreate2.udiStatus < 65534 THEN
							tylocalMcParam.Out.eStatus		:= Error;

							IF fbDirCreate2.udiStatus = 1908 THEN
								udiStatus	:= 10001;	//Create Machine Parameter Directory Error
							ELSE
								udiStatus	:= fbDirCreate2.udiStatus;
							END_IF
						END_IF

				END_CASE

			END_IF

		McParamActWrite:
			IF tylocalMcParam.Out.eStatus = Idle OR tylocalMcParam.Out.eStatus = Busy THEN

				tylocalMcParam.Out.eStatus	:= Busy;

				sStatTxt	:= a_sStatText[tylocalMcParam.Out.eStat];

				fbFileWrite1(bEn := TRUE);

				IF fbFileWrite1.udiStatus = 0 THEN
					tyMcParamCurr	:= tylocalMcParam.In.tyMcParmWr;
					tylocalMcParam.Out.eStatus			:= Done;
				ELSIF fbFileWrite1.udiStatus < 65534 THEN
					tylocalMcParam.Out.eStatus			:= Error;

					IF fbFileWrite1.udiStatus = 1900 THEN
						udiStatus	:= 10002;	//File Open Error While Writing
					ELSIF fbFileWrite1.udiStatus = 1901 THEN
						udiStatus	:= 10003;	//File Create Error While Writing
					ELSIF fbFileWrite1.udiStatus = 1903 THEN
						udiStatus	:= 10004;	//File Write Error
					ELSIF fbFileWrite1.udiStatus = 1904 THEN
						udiStatus	:= 10005;	//File Close Error While Writing
					ELSIF fbFileWrite1.udiStatus = 1914 THEN
						udiStatus	:= 10009;	//Directory Does Not Exist While Writing
					ELSE
						udiStatus	:= fbFileWrite1.udiStatus;
					END_IF
				END_IF

			END_IF

		McParamActRead:
			IF tylocalMcParam.Out.eStatus = Idle OR tylocalMcParam.Out.eStatus = Busy THEN

				tylocalMcParam.Out.eStatus	:= Busy;

				sStatTxt	:= a_sStatText[tylocalMcParam.Out.eStat];

				fbFileRead1(bEn := TRUE);
				IF fbFileRead1.udiStatus = 0 THEN
					tylocalMcParam.Out.eStatus			:= Done;
				ELSIF fbFileRead1.udiStatus < 65534 THEN
					tylocalMcParam.Out.eStatus		:= Error;

					IF fbFileRead1.udiStatus = 1900 THEN
						udiStatus	:= 10006;	//File Open Error While Reading
					ELSIF fbFileRead1.udiStatus = 1902 THEN
						udiStatus	:= 10007;	//File Read Error
					ELSIF fbFileRead1.udiStatus = 1904 THEN
						udiStatus	:= 10008;	//File Close Error While Reading
					ELSIF fbFileRead1.udiStatus = 1915 THEN
						tylocalMcParam.Out.eStatus			:= Done;
						bFileNotFound	:= TRUE;
					ELSE
						udiStatus	:= fbFileRead1.udiStatus;
					END_IF
				END_IF

			END_IF

	END_CASE

END_ACTION
```

#### Act_Alarm.st - Do Not Change!!!
```iecst
(** 2019-03-25 **)
ACTION Act_Alarm:

	IF tylocalMcParam.In.udiRstErr <> udiRstErrOld THEN
		bRstErr			:= TRUE;
		udiRstErrOld	:= tylocalMcParam.In.udiRstErr;
	ELSE
		bRstErr			:= FALSE;
	END_IF

	//Reset Error
	IF (tylocalMcParam.Out.eStatus = Error) AND bRstErr THEN
		tylocalMcParam.In.eAct	:= McParamActIdle;
		tylocalMcParam.Out.eStat	:= McParamActIdle;
	END_IF

	//Reset Done
	IF tylocalMcParam.Out.eStatus = Done AND tylocalMcParam.In.eAct = McParamActIdle THEN
		tylocalMcParam.Out.eStat	:= McParamActIdle;
	END_IF

	//Set p_eAct
	IF tylocalMcParam.Out.eStatus = Idle THEN
		tylocalMcParam.Out.eStat	:= tylocalMcParam.In.eAct;
	END_IF

	//Error
	IF EDGEPOS(tylocalMcParam.Out.eStatus = Error) THEN

		tylocalMcParam.Out.tyAlmData.sProgNm		:= g_tyNtParamCurr.sMcParamFileNm;
		tylocalMcParam.Out.tyAlmData.udiCode		:= udiStatus;
		tylocalMcParam.Out.tyAlmData.eSeverity		:= AlmSeverityError;
		tylocalMcParam.Out.tyAlmData.udiRunTime		:= tylocalMcParam.Out.tyAlmData.udiRunTime + 1;
		tylocalMcParam.Out.tyAlmData.bAlm			:= TRUE;
		tylocalMcParam.Out.tyAlmData.udiModuleNum  	:= udiModuleNum;
		g_sMcParamProgNm		:= g_tyNtParamCurr.sMcParamFileNm;

		//Get Error Message
		IF tylocalMcParam.Out.tyAlmData.udiCode < 10000 OR tylocalMcParam.Out.tyAlmData.udiCode > 10099 THEN
			tylocalMcParam.Out.tyAlmData.sAlmMsg	:= 'Unknown';
			tylocalMcParam.Out.tyAlmData.sRcyMsg	:= 'Unknown';
		ELSE
			tylocalMcParam.Out.tyAlmData.sAlmMsg	:= a_tyAlmText[tylocalMcParam.Out.tyAlmData.udiCode].sAlmText;
			tylocalMcParam.Out.tyAlmData.sRcyMsg	:= a_tyAlmText[tylocalMcParam.Out.tyAlmData.udiCode].sRcyText;
		END_IF

		tylocalMcParam.Out.sStatTxt	:= tylocalMcParam.Out.tyAlmData.sAlmMsg;
	ELSIF bConnected = FALSE THEN
		tylocalMcParam.Out.tyAlmData.sProgNm		:= g_tyNtParamCurr.sMcParamFileNm;
		tylocalMcParam.Out.tyAlmData.udiCode		:= udiStatus;
		tylocalMcParam.Out.tyAlmData.eSeverity		:= AlmSeverityWarning;
		tylocalMcParam.Out.tyAlmData.udiRunTime		:= tylocalMcParam.Out.tyAlmData.udiRunTime + 1;
		tylocalMcParam.Out.tyAlmData.bWarning		:= TRUE;
		tylocalMcParam.Out.tyAlmData.udiModuleNum 	:= udiModuleNum;
		g_sMcParamProgNm							:= g_tyNtParamCurr.sMcParamFileNm;

		//Get Error Message
		IF tylocalMcParam.Out.tyAlmData.udiCode < 10000 OR tylocalMcParam.Out.tyAlmData.udiCode > 10099 THEN
			tylocalMcParam.Out.tyAlmData.sAlmMsg	:= 'Unknown';
			tylocalMcParam.Out.tyAlmData.sRcyMsg	:= 'Unknown';
		ELSE
			tylocalMcParam.Out.tyAlmData.sAlmMsg	:= a_tyAlmText[tylocalMcParam.Out.tyAlmData.udiCode].sAlmText;
			tylocalMcParam.Out.tyAlmData.sRcyMsg	:= a_tyAlmText[tylocalMcParam.Out.tyAlmData.udiCode].sRcyText;
		END_IF

		tylocalMcParam.Out.sStatTxt	:= tylocalMcParam.Out.tyAlmData.sAlmMsg;
	ELSIF bRstErr AND (tylocalMcParam.Out.tyAlmData.udiCode <> 0) THEN

		tylocalMcParam.Out.tyAlmData.udiCode	:= 0;
		tylocalMcParam.Out.tyAlmData.eSeverity	:= AlmSeverityNA;
		tylocalMcParam.Out.tyAlmData.sAlmMsg	:= '';
		tylocalMcParam.Out.tyAlmData.sRcyMsg	:= '';
		tylocalMcParam.Out.tyAlmData.bAlm			:= FALSE;
		tylocalMcParam.Out.tyAlmData.bWarning		:= FALSE;
		tylocalMcParam.Out.sStatTxt	:= a_sStatText[tylocalMcParam.Out.eStat];

	END_IF

END_ACTION
```

#### Local.var - Do Not Change!!!
```iecst
(*2019-04-30*)
(**)
(*Local Action, State & Status*)
VAR
	tylocalMcParam : tyMcParamGen;
	eAct : eMcParamAction := McParamActIdle;
	eStat : eMcParamAction := McParamActIdle;
	eStatus : eFBStatus := Idle;
	udiStatus : UDINT := 0;
	sStatTxt : STRING[200] := '';
	a_sStatText : ARRAY[0..50] OF STRING[200] := ['Idling','Creating Directory','Reading Files','Writing Files',47('')];
END_VAR
(**)
(*Local Alarm*)
VAR
	tyAlmData : tyAlmDat;
	a_tyAlmText : ARRAY[10000..10099] OF tyAlmTxt := [(sAlmText:='Create User Directory Error',sRcyText:='Unable To Create User Directory. Please Contact Nutek For A Possible Solution'),(sAlmText:='Create Machine Parameter Directory Error',sRcyText:='Unable To Create Machine Parameter Directory. Please Contact Nutek For A Possible Solution'),(sAlmText:='File Open Error While Writing',sRcyText:='An Error Was Encountered While Trying To Open File. Please Contact Nutek For A Possible Solution.'),(sAlmText:='File Create Error While Writing',sRcyText:='An Error Was Encountered While Trying To Create File. Please Contact Nutek For A Possible Solution.'),(sAlmText:='File Write Error',sRcyText:='An Error Was Encountered While Trying To Write File. Please Contact Nutek For A Possible Solution.'),(sAlmText:='File Close Error While Writing',sRcyText:='An Error Was Encountered While Trying To Close File. Please Contact Nutek For A Possible Solution.'),(sAlmText:='File Open Error While Reading',sRcyText:='An Error Was Encountered While Trying To Open File. Please Contact Nutek For A Possible Solution.'),(sAlmText:='File Read Error',sRcyText:='An Error Was Encountered While Trying To Read File. Please Contact Nutek For A Possible Solution.'),(sAlmText:='File Close Error While Reading',sRcyText:='An Error Was Encountered While Trying To Close File. Please Contact Nutek For A Possible Solution.'),(sAlmText:='Directory Does Not Exist While Writing',sRcyText:='The Directory Does Not Exist.Please Contact Nutek For A Possibe Solution.'),90(0)];
END_VAR
(**)
(*Local Output*)
VAR
	tyMcParamCurr : tyMcParam;
	bFileNotFound : BOOL;
END_VAR
(**)
(*Local Input*)
VAR
	udiRstErr : UDINT := 0;
	sFileName : STRING[80] := 'MachineParameter.dat';
	tyMcParamWr : tyMcParam;
	sProgNm : STRING[15] := 'McParam';
	bNtSettingsLoadDone : BOOL := TRUE;
	bSvyHermesWriteConfig : BOOL;
END_VAR
(**)
(*Local*)
VAR
	bRstErr : BOOL;
	udiRstErrOld : UDINT;
	bInitDone : BOOL;
	bInitialDone : BOOL;
	usiStep : USINT;
	tyMcParamTemp : tyMcParam;
	fbDirCreate1 : fbDirCreate;
	fbDirCreate2 : fbDirCreate;
	fbFileRead1 : fbFileFullRead;
	fbFileWrite1 : fbFileFullWrite;
	fbFileWrite2 : fbFileFullWrite;
	udiModuleNum : UINT := 5251;
END_VAR
(*//ADD*)
VAR
	sHMIIPAddr : STRING[15];
	sVNCIPAddr : STRING[15];
	uiNSIdx : UINT;
	fbConnectOPCUA : fbOPCUAConnect;
	fbDisconnectOPCUA : fbOPCUADisconnect;
	dwConnectionHdl : DWORD;
	sHMIAddrNodeID : STRING[15];
	sVNCAddrNodeID : STRING[5];
	fbReadGetNodeHdlList : fbOPCUAGetNodeHdlList;
	fbReadList : fbOPCUAReadList;
	tyReadHdls : tyOPCUAHdlList;
	fbWriteGetNodeHdlList : fbOPCUAGetNodeHdlList;
	fbWriteList : fbOPCUAWriteList;
	tyWriteHdls : tyOPCUAHdlList;
	sObjIDNodeID : STRING[5];
	sSaveCfgNodeID : STRING[5];
	fbSaveCfgMethodGetHdl : fbOPCUAMethodGetHandle;
	fbSaveCfgMethodCall : fbOPCUAMethodCall;
	sLoadCfgNodeID : STRING[5];
	fbLoadCfgMethodGetHdl : fbOPCUAMethodGetHandle;
	fbLoadCfgMethodCall : fbOPCUAMethodCall;
	dwMethodHdl : DWORD;
	usiChkIpAddrStep : USINT;
	bWarning : BOOL;
	bConnected : BOOL;
END_VAR
```

#### InputRef.var - not listed in the package file held
```iecst
(*2019-03-25*)
(**)
(*General*)
VAR
	p_eAct : REFERENCE TO eMcParamAction;
	p_udiRstErr : REFERENCE TO UDINT;
END_VAR
(**)
(*Configuration*)
VAR
	p_sFileName : REFERENCE TO STRING[80];
	p_tyMcParamWr : REFERENCE TO tyMcParam;
	p_sProgNm : REFERENCE TO STRING[15];
	p_bNtSettingsLoadDone : REFERENCE TO BOOL;
	p_bRmtHermesWriteConfig : REFERENCE TO BOOL;
	p_bSvyHermesWriteConfig : REFERENCE TO BOOL;
	p_tyHermesConfigurationWr : REFERENCE TO tyHermesConfiguration;
	p_bNtParamAutoRcpPrep : REFERENCE TO BOOL;
	p_bNtParamProjLaneBPrep : REFERENCE TO BOOL;
	p_eNtParamCustomerReq : REFERENCE TO eCustomer;
	p_eNtParamAutoRcpPrecededBy : REFERENCE TO eAutoRcpPreceded;
END_VAR
(*//ADD*)
VAR
	p_sHWInfoIPAddr : REFERENCE TO STRING[15];
	p_sUISetHMIIPAddr : REFERENCE TO STRING[15];
	p_bAlarmWarning : REFERENCE TO BOOL;
	p_bUIUpdtHMIIPAddr : REFERENCE TO BOOL;
END_VAR
```

#### Act_InitGlobal.st - not listed in the package file held
```iecst
(** 2019-03-25 **)
ACTION Act_InitGlobal:

	(* Always Change If Project Change *)

	//Pass Data To Link
	p_bLinkStartupRun ACCESS p_StartupRun;

	//Pass Data To Internal Use
	p_udiRstErr ACCESS p_RstErrReset;
	p_sFileName ACCESS p_NtParamMcParamFileNm;
	p_tyMcParamWr ACCESS p_UIMcParamWr;
	p_sProgNm ACCESS p_NtParamMcParamProgNm;
	p_bNtSettingsLoadDone ACCESS p_StartupNtSettingsLoadDone;
	p_bRmtHermesWriteConfig ACCESS p_RmtHermesWriteConfig; //new for Hermes 1.3
	p_bSvyHermesWriteConfig ACCESS p_SvyHermesWriteConfig; //new for Hermes 1.3
	p_tyHermesConfigurationWr ACCESS p_HermesConfigurationWr; //new for Hermes 1.3
	//Controling AutoRcp
	p_bNtParamAutoRcpPrep ACCESS p_NtParamAutoRcpPrep;
	p_bNtParamProjLaneBPrep ACCESS p_NtParamProjLaneBPrep;
	p_eNtParamCustomerReq ACCESS p_NtParamCustomerReq;
	p_eNtParamAutoRcpPrecededBy ACCESS p_NtParamAutoRcpPrecededBy;
	(* Always Change If Project Change *)
	//ADD
	p_sUISetHMIIPAddr ACCESS p_UISetHMIIPAddr;
	p_sHWInfoIPAddr ACCESS p_HWInfoIPAddr;
	p_bUIUpdtHMIIPAddr ACCESS p_UIUpdtHMIIPAddr;
	p_bAlarmWarning ACCESS p_AlarmWarning;
END_ACTION
```

#### Act_InitLocal.st - not listed in the package file held
```iecst
(** 2019-03-25 **)
ACTION Act_InitLocal:

	//Input Reference Link To Local Variable
	p_eAct ACCESS ADR(eAct);
	p_udiRstErr ACCESS ADR(udiRstErr);
	p_sFileName ACCESS ADR(sFileName);
	p_tyMcParamWr ACCESS ADR(tyMcParamWr);
	p_sProgNm ACCESS ADR(sProgNm);
	p_bNtSettingsLoadDone ACCESS ADR(bNtSettingsLoadDone);
	p_bSvyHermesWriteConfig ACCESS ADR(bSvyHermesWriteConfig);

	//ADD
	p_bAlarmWarning ACCESS ADR(bWarning);
END_ACTION
```

#### Act_LinkAction.st - not listed in the package file held
```iecst
(** 2019-03-29 **)
ACTION Act_LinkAction:

	IF p_bLinkStartupRun = TRUE THEN
		p_eAct ACCESS p_StartupMcParamAct;
	ELSIF p_bSvyHermesWriteConfig THEN 	//new for Hermes 1.3
		p_eAct ACCESS p_SvyHermesMcParamAct; //Changed
	ELSIF p_bRmtHermesWriteConfig THEN 	//new for Hermes 1.3
		p_eAct ACCESS p_RmtHermesMcParamAct;
	ELSE
		p_eAct ACCESS p_UIMcParamAct;
	END_IF

END_ACTION
```

#### Init.st - not listed in the package file held
```iecst
(** 2020-09-22 **)
PROGRAM _INIT

	(* Always Change If Project Change *)

	//Pass Address To Global Address For External Use
	//Action, State & Status
	p_McParamStat		:= ADR(eStat);
	p_McParamStatus		:= ADR(eStatus);
	p_McParamStatTxt	:= ADR(sStatTxt);

	//Alarmhorizontal
	p_McParamAlmData	:= ADR(tyAlmData);

	//Output
	p_McParamFileNotFound				:= ADR(bFileNotFound);

	p_McParamCurr						:= ADR(tyMcParamCurr);

	p_McParamLFOnline					:= ADR(tyMcParamCurr.a_bLFOnline);
	p_McParamLFIPAddr					:= ADR(tyMcParamCurr.a_sLFIPAddr);

	p_McParamMcNm						:= ADR(tyMcParamCurr.sMcNm);
	p_McParamSSaverTm					:= ADR(tyMcParamCurr.uiSSaverTmInSec);
	p_McParamSSaverEn					:= ADR(tyMcParamCurr.bSSaverEn);
	p_McParamDefaultMcMod				:= ADR(tyMcParamCurr.usiDefaultMcMod);
	p_McParamWidthAtHmPos				:= ADR(tyMcParamCurr.diWidthAtHmPosInUM);
	p_McParamConvInitTm					:= ADR(tyMcParamCurr.diConvInitTmInMS);
	p_McParamTranInErrDlyTm				:= ADR(tyMcParamCurr.diTranInErrDlyTmInMS);
	p_McParamMag1ConvRunTmOut			:= ADR(tyMcParamCurr.diMag1ConvRunTmOutInMS);
	p_McParamMag2ConvRunTmOut			:= ADR(tyMcParamCurr.diMag2ConvRunTmOutInMS);
	p_McParamMag3ConvRunTmOut			:= ADR(tyMcParamCurr.diMag3ConvRunTmOutInMS);
	p_McParamOvenMaxBffr				:= ADR(tyMcParamCurr.diOvenMaxBffr);
	p_McParamTravPosA					:= ADR(tyMcParamCurr.diTravPosA);
	p_McParamTravPosB					:= ADR(tyMcParamCurr.diTravPosB);
	p_McParamLifterPosA					:= ADR(tyMcParamCurr.diLifterPosA);
	p_McParamLifterPosB					:= ADR(tyMcParamCurr.diLifterPosB);
	p_McParamAWDis						:= ADR(tyMcParamCurr.bAWDis);
	p_McParamMnlAccDat					:= ADR(tyMcParamCurr.bMnlAccDat);
	p_McParamAutoStepEn					:= ADR(tyMcParamCurr.bAutoStepEn);
	p_McParamVSMEMAEn					:= ADR(tyMcParamCurr.bVSMEMAEn);
	p_McParamChgParamEn					:= ADR(tyMcParamCurr.bChgParamEn);
	p_McParamHermesRmtEn				:= ADR(tyMcParamCurr.bHermesRmtEn);
	p_McParamGapBwtnBrdEn				:= ADR(tyMcParamCurr.bGapBwtnBrdEn);
	p_McParamLongBrdEn					:= ADR(tyMcParamCurr.bLongBrdEn);
	p_McParamOvenEn						:= ADR(tyMcParamCurr.bOvenEn);
	p_McParamExtdOvenEn					:= ADR(tyMcParamCurr.bExtdOvenEn);
	p_McParamInShutterDis				:= ADR(tyMcParamCurr.bInShutterDis);
	p_McParamStopperADis				:= ADR(tyMcParamCurr.bStopperADis);
	p_McParamStopperBDis				:= ADR(tyMcParamCurr.bStopperBDis);
	p_McParamMagAutoDetTm				:= ADR(tyMcParamCurr.diMagAutoDetectSenTmInMS);
	p_McParamAGVComEn					:= ADR(tyMcParamCurr.bAGVComEn);

	p_McParamLFEn						:= ADR(tyMcParamCurr.bLFEn);
	p_McParamLCSLFEn					:= ADR(tyMcParamCurr.bLCSLFEn);
	p_McParamLCSReqRcpEn				:= ADR(tyMcParamCurr.bLCSReqRcpEn);
	p_McParamLCSManageRcpEn				:= ADR(tyMcParamCurr.bLCSManageRcpEn);
	p_McParamLCSLiveDatEn				:= ADR(tyMcParamCurr.bLCSLiveDatEn);
	p_McParamLFLeaderMc					:= ADR(tyMcParamCurr.bLFLeaderMc);
	p_McParamSectionLeader				:= ADR(tyMcParamCurr.bSectionLeader);
	p_McParamUSWidthChkEn				:= ADR(tyMcParamCurr.bUSWidthChkEn);
	p_McParamLFMcIdxBeforeOven			:= ADR(tyMcParamCurr.diLFMcIdxBeforeOven);
	p_McParamLFMcIdxAfterOven			:= ADR(tyMcParamCurr.diLFMcIdxAfterOven);

	p_McParamLang						:= ADR(tyMcParamCurr.usiLang);

	p_McParamConvLftSenAntiGap			:= ADR(tyMcParamCurr.tyLftSenAntiGapDly);
	p_McParamConvLftSenOnTm				:= ADR(tyMcParamCurr.tyLftSenAntiGapDly.diSigOnTm);
	p_McParamConvLftSenOffTm			:= ADR(tyMcParamCurr.tyLftSenAntiGapDly.diSigOffTm);
	p_McParamConvMidSenAntiGap			:= ADR(tyMcParamCurr.tyMidSenAntiGapDly);
	p_McParamConvMidSenOnTm				:= ADR(tyMcParamCurr.tyMidSenAntiGapDly.diSigOnTm);
	p_McParamConvMidSenOffTm			:= ADR(tyMcParamCurr.tyMidSenAntiGapDly.diSigOffTm);
	p_McParamConvRgtSenAntiGap			:= ADR(tyMcParamCurr.tyRgtSenAntiGapDly);
	p_McParamConvRgtSenOnTm				:= ADR(tyMcParamCurr.tyRgtSenAntiGapDly.diSigOnTm);
	p_McParamConvRgtSenOffTm			:= ADR(tyMcParamCurr.tyRgtSenAntiGapDly.diSigOffTm);
	p_McParamConvClrSenAntGap			:= ADR(tyMcParamCurr.tyClrSenAntiGapDly);
	p_McParamConvClrSenOnTm				:= ADR(tyMcParamCurr.tyClrSenAntiGapDly.diSigOnTm);
	p_McParamConvClrSenOffTm			:= ADR(tyMcParamCurr.tyClrSenAntiGapDly.diSigOffTm);

	p_McParamMagConvEntrySenAntiGap		:= ADR(tyMcParamCurr.tyMagConvEntrySenAntiGapDly);
	p_McParamMagConvEntrySenOnTm		:= ADR(tyMcParamCurr.tyMagConvEntrySenAntiGapDly.diSigOnTm);
	p_McParamMagConvEntrySenOffTm		:= ADR(tyMcParamCurr.tyMagConvEntrySenAntiGapDly.diSigOffTm);

	p_McParamMagConvPresentAntiGap		:= ADR(tyMcParamCurr.tyMagConvPresentSenAntiGapDly);
	p_McParamMagConvPresentSenOnTm		:= ADR(tyMcParamCurr.tyMagConvPresentSenAntiGapDly.diSigOnTm);
	p_McParamMagConvPresentSenOffTm		:= ADR(tyMcParamCurr.tyMagConvPresentSenAntiGapDly.diSigOffTm);

	p_McParamUSCommAMod					:= ADR(tyMcParamCurr.eUSCommA);
	p_McParamUSSMEMAAParam				:= ADR(tyMcParamCurr.tyUSCommASMEMA);
	p_McParamUSSMEMAASelection			:= ADR(tyMcParamCurr.tyUSCommASMEMA.eSelection);
	p_McParamUBAAStatSetGd				:= ADR(tyMcParamCurr.tyUSCommASMEMA.bStatSigSetGd);

	p_McParamUSCommBMod					:= ADR(tyMcParamCurr.eUSCommB);
	p_McParamUSSMEMABParam				:= ADR(tyMcParamCurr.tyUSCommBSMEMA);
	p_McParamUSSMEMABSelection			:= ADR(tyMcParamCurr.tyUSCommBSMEMA.eSelection);
	p_McParamUBABStatSetGd				:= ADR(tyMcParamCurr.tyUSCommBSMEMA.bStatSigSetGd);

	p_McParamLFMcIdxBeforeOven2			:= ADR(tyMcParamCurr.diLFMcIdxBeforeOven2);
	p_McParamLFMcIdxAfterOven2			:= ADR(tyMcParamCurr.diLFMcIdxAfterOven2);
	//	p_McParamAIVComm					:= ADR(tyMcParamCurr.tyAIVComm);
	//	p_McParamAIVSvrPort					:= ADR(tyMcParamCurr.tyAIVComm.uiSvrPort);
	//	p_McParamAIVClientPort				:= ADR(tyMcParamCurr.tyAIVComm.uiClientPort);
	//	p_McParamAIVClientAddr				:= ADR(tyMcParamCurr.tyAIVComm.sClientAddress);

	p_McParamWidthOffset				:= ADR(tyMcParamCurr.diWidthOffsetInUM);

	p_McParamNetworkMod					:= ADR(tyMcParamCurr.eNetworkMod);

	p_McParamLFSeqStayActive			:= ADR(tyMcParamCurr.bLFSeqStayActive);

	p_McParamMagAWDis					:= ADR(tyMcParamCurr.bMagAWDis);
	p_McParamMagSafetyBarDis			:= ADR(tyMcParamCurr.bMagSafetyBarDis);
	p_McParamMag1WidthAtHmPos			:= ADR(tyMcParamCurr.diMag1WidthAtHmPosInUM);
	p_McParamMag2WidthAtHmPos			:= ADR(tyMcParamCurr.diMag2WidthAtHmPosInUM);
	p_McParamMag3WidthAtHmPos			:= ADR(tyMcParamCurr.diMag3WidthAtHmPosInUM);
	p_McParamLFBuzMute					:= ADR(tyMcParamCurr.bLFBuzMute);

	p_McParamAGVComProtocol				:= ADR(tyMcParamCurr.eAGVComProtocol);
	p_McParamMagExMode					:= ADR(tyMcParamCurr.eMagExMode);

	p_McParamAWPusherAtHmPos			:= ADR(tyMcParamCurr.diAWPusherAtHmPosInUM);
	p_McParamAWPusherDis				:= ADR(tyMcParamCurr.bAWPusherDis);

	p_McParamTravInletFixtoFixPos	:= ADR(tyMcParamCurr.diTravInletFixtoFixPos);
	p_McParamDisableFMWarning		:= ADR(tyMcParamCurr.bDisableFMWarning);

	p_McParamConvLineAInletSenOnTm	:= ADR(tyMcParamCurr.tyLineAInletSenAntiGapDly.diSigOnTm);
	p_McParamConvLineAInletSenOffTm	:= ADR(tyMcParamCurr.tyLineAInletSenAntiGapDly.diSigOffTm);
	p_McParamConvLineBInletSenOnTm	:= ADR(tyMcParamCurr.tyLineBInletSenAntiGapDly.diSigOnTm);
	p_McParamConvLineBInletSenOffTm	:= ADR(tyMcParamCurr.tyLineBInletSenAntiGapDly.diSigOffTm);
	p_McParamUSWidthChkSenOnTm		:= ADR(tyMcParamCurr.tyUSWidthChkSenAntiGapDly.diSigOnTm);
	p_McParamUSWidthChkSenOffTm		:= ADR(tyMcParamCurr.tyUSWidthChkSenAntiGapDly.diSigOffTm);

	p_McParamDBAOnWOAlign			:= ADR(tyMcParamCurr.bDBAOnWOAlign);

	//MagConv top and bottom
	p_McParamInMagConvEntSenOnTm	:= ADR(tyMcParamCurr.tyInMagConvEntAntiGapDly.diSigOnTm);
	p_McParamInMagConvEntSenOffTm	:= ADR(tyMcParamCurr.tyInMagConvEntAntiGapDly.diSigOffTm);
	p_McParamInMagConvExtSenOnTm	:= ADR(tyMcParamCurr.tyInMagConvExtAntiGapDly.diSigOnTm);
	p_McParamInMagConvExtSenOffTm	:= ADR(tyMcParamCurr.tyInMagConvExtAntiGapDly.diSigOffTm);
	p_McParamInMagConvMidSenOnTm	:= ADR(tyMcParamCurr.tyInMagConvMidAntiGapDly.diSigOnTm);
	p_McParamInMagConvMidSenOffTm	:= ADR(tyMcParamCurr.tyInMagConvMidAntiGapDly.diSigOffTm);

	p_McParamOutMagConvEntSenOnTm	:= ADR(tyMcParamCurr.tyOutMagConvEntAntiGapDly.diSigOnTm);
	p_McParamOutMagConvEntSenOffTm	:= ADR(tyMcParamCurr.tyOutMagConvEntAntiGapDly.diSigOffTm);
	p_McParamOutMagConvExtSenOnTm	:= ADR(tyMcParamCurr.tyOutMagConvExtAntiGapDly.diSigOnTm);
	p_McParamOutMagConvExtSenOffTm	:= ADR(tyMcParamCurr.tyOutMagConvExtAntiGapDly.diSigOffTm);
	p_McParamOutMagConvMidSenOnTm	:= ADR(tyMcParamCurr.tyOutMagConvMidAntiGapDly.diSigOnTm);
	p_McParamOutMagConvMidSenOffTm	:= ADR(tyMcParamCurr.tyOutMagConvMidAntiGapDly.diSigOffTm);

	p_McParamInMagConv2EntSenOnTm	:= ADR(tyMcParamCurr.tyInMagConv2EntAntiGapDly.diSigOnTm);
	p_McParamInMagConv2EntSenOffTm	:= ADR(tyMcParamCurr.tyInMagConv2EntAntiGapDly.diSigOffTm);
	p_McParamInMagConv2ExtSenOnTm	:= ADR(tyMcParamCurr.tyInMagConv2ExtAntiGapDly.diSigOnTm);
	p_McParamInMagConv2ExtSenOffTm	:= ADR(tyMcParamCurr.tyInMagConv2ExtAntiGapDly.diSigOffTm);
	p_McParamInMagConv2MidSenOnTm	:= ADR(tyMcParamCurr.tyInMagConv2MidAntiGapDly.diSigOnTm);
	p_McParamInMagConv2MidSenOffTm	:= ADR(tyMcParamCurr.tyInMagConv2MidAntiGapDly.diSigOffTm);

	p_McParamOutMagConv2EntSenOnTm	:= ADR(tyMcParamCurr.tyOutMagConv2EntAntiGapDly.diSigOnTm);
	p_McParamOutMagConv2EntSenOffTm	:= ADR(tyMcParamCurr.tyOutMagConv2EntAntiGapDly.diSigOffTm);
	p_McParamOutMagConv2ExtSenOnTm	:= ADR(tyMcParamCurr.tyOutMagConv2ExtAntiGapDly.diSigOnTm);
	p_McParamOutMagConv2ExtSenOffTm	:= ADR(tyMcParamCurr.tyOutMagConv2ExtAntiGapDly.diSigOffTm);
	p_McParamOutMagConv2MidSenOnTm	:= ADR(tyMcParamCurr.tyOutMagConv2MidAntiGapDly.diSigOnTm);
	p_McParamOutMagConv2MidSenOffTm	:= ADR(tyMcParamCurr.tyOutMagConv2MidAntiGapDly.diSigOffTm);

	p_McParamInMagConvRunTmOut		:= ADR(tyMcParamCurr.diInMagConvRunTmOutInMS);
	p_McParamOutMagConvRunTmOut		:= ADR(tyMcParamCurr.diOutMagConvRunTmOutInMS);
	p_McParamLifterMagConvRunTmOut	:= ADR(tyMcParamCurr.diLifterMagConvRunTmOutInMS);
	p_McParamInMagConv2RunTmOut		:= ADR(tyMcParamCurr.diInMagConv2RunTmOutInMS);
	p_McParamOutMagConv2RunTmOut	:= ADR(tyMcParamCurr.diOutMagConv2RunTmOutInMS);
	p_McParamLifterMagConv2RunTmOut	:= ADR(tyMcParamCurr.diLifterMagConv2RunTmOutInMS);
	p_McParamLifterTopPos			:= ADR(tyMcParamCurr.diLifterTopPos);
	p_McParamLifterBtmPos			:= ADR(tyMcParamCurr.diLifterBtmPos);
	p_McParamLifterTopPos2			:= ADR(tyMcParamCurr.diLifterTopPos2);
	p_McParamLifterBtmPos2			:= ADR(tyMcParamCurr.diLifterBtmPos2);
	p_McParamTCPSvrPort				:= ADR(tyMcParamCurr.diTCPSvrPort);
	p_McParamMagWidthChkDis			:= ADR(tyMcParamCurr.bMagWidthChkDis);
	p_McParamMag1WidthChkDetDist	:= ADR(tyMcParamCurr.diMag1WidthChkDetDist);
	p_McParamMag2WidthChkDetDist	:= ADR(tyMcParamCurr.diMag2WidthChkDetDist);
	p_McParamMag3WidthChkDetDist	:= ADR(tyMcParamCurr.diMag3WidthChkDetDist);
	p_McParamTopScannerEn			:= ADR(tyMcParamCurr.bTopScannerEn);
	p_McParamBtmScannerEn			:= ADR(tyMcParamCurr.bBtmScannerEn);
	p_McParamTopScanIP				:= ADR(tyMcParamCurr.sTopScanIPAddr);
	p_McParamTopScanPort			:= ADR(tyMcParamCurr.uiTopScanSvrPort);
	p_McParamBtmScanIP				:= ADR(tyMcParamCurr.sBtmScanIPAddr);
	p_McParamBtmScanPort			:= ADR(tyMcParamCurr.uiBtmScanSvrPort);
	p_McParamOpConEn				:= ADR(tyMcParamCurr.bOpConEn);
	p_McParamOpConIP				:= ADR(tyMcParamCurr.sOpConIPAddr);
	p_McParamOpConPort				:= ADR(tyMcParamCurr.uiOpConSvrPort);
	p_McParamOpConParam				:= ADR(tyMcParamCurr.tyOpConParam);

	p_McParamSiemensPrep            := ADR(tyMcParamCurr.bSiemensPrep);  //ADD
	p_McParamHermesSvyEn			:= ADR(tyMcParamCurr.bHermesSvyEn);//new for Hermes 1.3
	p_McParamHermesScannerEn		:= ADR(tyMcParamCurr.bHermesScannerEn);//new for Hermes 1.3
	//Siemen
	p_McParamInStopperDis			:= ADR(tyMcParamCurr.bInStopperDis);
	p_McParamInStopperExtDelayTm	:= ADR(tyMcParamCurr.diInletStopperExtDelayTmInMS);
	p_McParamMESEn					:= ADR(tyMcParamCurr.bMESEn); //bMESRFIDDis
	p_McParamMESResponseTO			:= ADR(tyMcParamCurr.diMESResponseTOTmInMS);
	p_McParamSwitchingProdType		:= ADR(tyMcParamCurr.bSwitchingProdType);
	p_McParamAutoRcpDisable 		:= ADR(tyMcParamCurr.bAutoRcpDisable); //Self Selected
	p_McParamAutoRcpBatchIDChgCmp	:= ADR(tyMcParamCurr.bBatchIDChgOverCmp);
	p_McParamAutoRcpIgnoreBtmClr	:= ADR(tyMcParamCurr.bIgnoreBtmClearance);
	p_McParamAutoRcpIgnoreTopClr	:= ADR(tyMcParamCurr.bIgnoreTopClearance);
	p_McParamAutoRcpIgnoreThickns	:= ADR(tyMcParamCurr.bIgnoreThickness);
	//DMC Scanner
	p_McParamDMCScannerEn			:= ADR(tyMcParamCurr.bDMCScannerEn);
	p_McParamDMCScanWriteTO			:= ADR(tyMcParamCurr.diDMCScanTOErrInMs);

	p_McParamDefaultGateway			:= ADR(tyMcParamCurr.sDefaultGateWay);//

	(* Always Change If Project Change *)

END_PROGRAM
```
